SPLINE
SPL {X  -124.075, Y  +778.932, Z    +0.000, E1   -61.393, E3 +52956.323}
SPL {X  -150.653, Y  +735.257, Z    +0.000, E1   -50.160, E3 +52964.002}
SPL {X  -159.377, Y  +706.804, Z    +0.000, E1   -34.828, E3 +52965.646}
SPL {X  -162.134, Y  +688.425, Z    +0.000, E1   -19.100, E3 +52965.583}
SPL {X  -162.803, Y  +675.871, Z    +0.000, E1    -5.469, E3 +52965.766}
SPL {X  -162.820, Y  +671.500, Z    +0.000, E1    +0.000, E3 +52965.335}
SPL {X  -162.820, Y  +669.743, Z    +0.000, E1    +4.352, E3 +52965.130}
SPL {X  -162.820, Y  +665.917, Z    +0.000, E1   +15.272, E3 +52965.125}
SPL {X  -162.820, Y  +659.880, Z    +0.000, E1   +32.256, E3 +52965.036}
SPL {X  -162.820, Y  +652.069, Z    +0.000, E1   +49.663, E3 +52965.062}
SPL {X  -162.820, Y  +641.345, Z    +0.000, E1   +63.138, E3 +52965.160}
SPL {X  -162.820, Y  +620.039, Z    +0.000, E1   +75.979, E3 +52963.770}
SPL {X  -162.820, Y  +571.094, Z    +0.000, E1   +77.089, E3 +52978.948}
SPL {X  -157.487, Y  +339.169, Z    +0.000, E1   +76.425, E3 +53072.052}
SPL {X  -156.386, Y  +335.181, Z    +0.000, E1   +75.555, E3 +53084.113}
SPL {X  -152.710, Y  +324.020, Z    +0.000, E1   +75.365, E3 +53091.924}
SPL {X  -139.497, Y  +296.529, Z    +0.000, E1   +77.231, E3 +53085.495}
ENDSPLINE

SPLINE
SPL {X  -139.520, Y  +296.568, Z    +0.000, E1   +75.884, E3 +53098.143}
ENDSPLINE

SPLINE
SPL {X  -138.554, Y  +294.984, Z    +0.000, E1   +74.772, E3 +53108.024}
SPL {X  -137.186, Y  +292.805, Z    +0.000, E1   +73.993, E3 +53115.264}
SPL {X  -133.270, Y  +286.961, Z    +0.000, E1   +73.739, E3 +53119.977}
SPL {X  -129.057, Y  +281.230, Z    +0.000, E1   +73.118, E3 +53126.885}
SPL {X  -123.859, Y  +274.815, Z    +0.000, E1   +72.511, E3 +53133.269}
SPL {X  -121.018, Y  +271.573, Z    +0.000, E1   +72.049, E3 +53136.787}
SPL {X  -113.980, Y  +264.229, Z    +0.000, E1   +74.120, E3 +53132.365}
SPL {X   -56.216, Y  +227.692, Z    +0.000, E1   +56.267, E3 +53309.089}
ENDSPLINE

SPLINE
SPL {X  -126.995, Y  +278.604, Z    +0.000, E1   +59.937, E3 +53481.329}
SPL {X  -150.196, Y  +317.640, Z    +0.000, E1   +49.956, E3 +53489.784}
SPL {X  -157.261, Y  +338.316, Z    +0.000, E1   +40.017, E3 +53491.479}
SPL {X  -160.924, Y  +355.726, Z    +0.000, E1   +27.715, E3 +53491.920}
SPL {X  -162.423, Y  +369.141, Z    +0.000, E1   +15.207, E3 +53492.356}
SPL {X  -162.811, Y  +378.755, Z    +0.000, E1    +4.616, E3 +53492.270}
SPL {X  -162.820, Y  +382.684, Z    +0.000, E1    -0.227, E3 +53491.825}
SPL {X  -162.820, Y  +385.721, Z    +0.000, E1    -8.371, E3 +53491.640}
SPL {X  -162.820, Y  +388.532, Z    +0.000, E1   -16.412, E3 +53491.527}
SPL {X  -162.820, Y  +392.558, Z    +0.000, E1   -27.778, E3 +53491.616}
SPL {X  -162.820, Y  +400.474, Z    +0.000, E1   -46.251, E3 +53491.479}
SPL {X  -162.820, Y  +414.510, Z    +0.000, E1   -65.115, E3 +53490.922}
SPL {X  -162.820, Y  +465.064, Z    +0.000, E1   -76.269, E3 +53500.770}
SPL {X  -157.184, Y  +715.968, Z    +0.000, E1   -76.600, E3 +53596.728}
SPL {X  -156.461, Y  +718.560, Z    +0.000, E1   -75.553, E3 +53610.148}
SPL {X  -153.015, Y  +729.150, Z    +0.000, E1   -75.312, E3 +53618.237}
SPL {X  -149.053, Y  +739.025, Z    +0.000, E1   -74.952, E3 +53627.033}
SPL {X  -144.053, Y  +749.389, Z    +0.000, E1   -74.457, E3 +53637.024}
SPL {X  -139.539, Y  +757.399, Z    +0.000, E1   -73.892, E3 +53645.731}
SPL {X  -136.017, Y  +762.997, Z    +0.000, E1   -73.579, E3 +53650.913}
SPL {X  -133.089, Y  +767.296, Z    +0.000, E1   -73.251, E3 +53655.371}
SPL {X  -129.985, Y  +771.553, Z    +0.000, E1   -72.801, E3 +53660.365}
SPL {X  -126.581, Y  +775.909, Z    +0.000, E1   -72.426, E3 +53664.676}
SPL {X  -123.329, Y  +779.803, Z    +0.000, E1   -71.936, E3 +53669.058}
SPL {X  -119.291, Y  +784.315, Z    +0.000, E1   -72.148, E3 +53670.470}
SPL {X   -57.587, Y  +825.796, Z    +0.000, E1   -56.753, E3 +53824.233}
ENDSPLINE

SPLINE
SPL {X  -124.075, Y  +778.932, Z    +0.000, E1   -61.393, E3 +54017.862}
SPL {X  -150.653, Y  +735.257, Z    +0.000, E1   -50.160, E3 +54025.541}
SPL {X  -159.377, Y  +706.804, Z    +0.000, E1   -34.828, E3 +54027.184}
SPL {X  -162.134, Y  +688.425, Z    +0.000, E1   -19.100, E3 +54027.121}
SPL {X  -162.803, Y  +675.871, Z    +0.000, E1    -5.469, E3 +54027.305}
SPL {X  -162.820, Y  +671.500, Z    +0.000, E1    +0.000, E3 +54026.873}
SPL {X  -162.820, Y  +669.743, Z    +0.000, E1    +4.352, E3 +54026.669}
SPL {X  -162.820, Y  +665.917, Z    +0.000, E1   +15.272, E3 +54026.663}
SPL {X  -162.820, Y  +659.880, Z    +0.000, E1   +32.256, E3 +54026.575}
SPL {X  -162.820, Y  +652.069, Z    +0.000, E1   +49.663, E3 +54026.600}
SPL {X  -162.820, Y  +641.345, Z    +0.000, E1   +63.138, E3 +54026.698}
SPL {X  -162.820, Y  +620.039, Z    +0.000, E1   +75.979, E3 +54025.308}
SPL {X  -162.820, Y  +578.479, Z    +0.000, E1   +77.260, E3 +54037.579}
SPL {X  -162.820, Y  +557.052, Z    +0.000, E1   +76.772, E3 +54046.060}
SPL {X  -157.487, Y  +339.169, Z    +0.000, E1   +76.425, E3 +54133.591}
SPL {X  -156.386, Y  +335.181, Z    +0.000, E1   +75.555, E3 +54145.652}
SPL {X  -152.710, Y  +324.020, Z    +0.000, E1   +75.365, E3 +54153.462}
SPL {X  -139.497, Y  +296.529, Z    +0.000, E1   +77.231, E3 +54147.034}
ENDSPLINE

SPLINE
SPL {X  -139.792, Y  +297.022, Z    +0.000, E1   +76.273, E3 +54155.729}
ENDSPLINE

SPLINE
SPL {X  -138.933, Y  +295.600, Z    +0.000, E1   +75.173, E3 +54166.212}
SPL {X  -137.186, Y  +292.805, Z    +0.000, E1   +73.993, E3 +54176.802}
SPL {X  -133.270, Y  +286.961, Z    +0.000, E1   +73.739, E3 +54181.515}
SPL {X  -130.283, Y  +282.844, Z    +0.000, E1   +73.297, E3 +54186.407}
SPL {X  -126.880, Y  +278.461, Z    +0.000, E1   +72.855, E3 +54191.158}
SPL {X  -124.135, Y  +275.140, Z    +0.000, E1   +72.554, E3 +54194.286}
SPL {X  -121.687, Y  +272.322, Z    +0.000, E1   +72.100, E3 +54197.765}
SPL {X  -113.980, Y  +264.229, Z    +0.000, E1   +74.120, E3 +54193.903}
SPL {X   -56.216, Y  +227.692, Z    +0.000, E1   +56.267, E3 +54370.627}
ENDSPLINE

SPLINE
SPL {X  -126.995, Y  +278.604, Z    +0.000, E1   +59.937, E3 +54542.868}
SPL {X  -150.196, Y  +317.640, Z    +0.000, E1   +49.956, E3 +54551.323}
SPL {X  -157.261, Y  +338.316, Z    +0.000, E1   +40.017, E3 +54553.018}
SPL {X  -160.924, Y  +355.726, Z    +0.000, E1   +27.715, E3 +54553.459}
SPL {X  -162.423, Y  +369.141, Z    +0.000, E1   +15.207, E3 +54553.894}
SPL {X  -162.811, Y  +378.755, Z    +0.000, E1    +4.616, E3 +54553.808}
SPL {X  -162.820, Y  +382.684, Z    +0.000, E1    -0.227, E3 +54553.363}
SPL {X  -162.820, Y  +385.721, Z    +0.000, E1    -8.371, E3 +54553.179}
SPL {X  -162.820, Y  +388.532, Z    +0.000, E1   -16.412, E3 +54553.065}
SPL {X  -162.820, Y  +392.558, Z    +0.000, E1   -27.778, E3 +54553.154}
SPL {X  -162.820, Y  +400.474, Z    +0.000, E1   -46.251, E3 +54553.018}
SPL {X  -162.820, Y  +414.510, Z    +0.000, E1   -65.115, E3 +54552.461}
SPL {X  -162.820, Y  +465.064, Z    +0.000, E1   -76.269, E3 +54562.309}
SPL {X  -157.184, Y  +715.968, Z    +0.000, E1   -76.600, E3 +54658.266}
SPL {X  -156.461, Y  +718.560, Z    +0.000, E1   -75.553, E3 +54671.686}
SPL {X  -151.911, Y  +732.096, Z    +0.000, E1   -75.235, E3 +54682.240}
SPL {X  -146.569, Y  +744.407, Z    +0.000, E1   -74.677, E3 +54694.044}
SPL {X  -142.375, Y  +752.491, Z    +0.000, E1   -74.335, E3 +54701.072}
SPL {X  -139.539, Y  +757.399, Z    +0.000, E1   -73.892, E3 +54707.269}
SPL {X  -136.017, Y  +762.997, Z    +0.000, E1   -73.579, E3 +54712.452}
SPL {X  -133.089, Y  +767.296, Z    +0.000, E1   -73.251, E3 +54716.910}
SPL {X  -129.985, Y  +771.553, Z    +0.000, E1   -72.801, E3 +54721.904}
SPL {X  -126.581, Y  +775.909, Z    +0.000, E1   -72.426, E3 +54726.215}
SPL {X  -123.329, Y  +779.803, Z    +0.000, E1   -71.936, E3 +54730.597}
SPL {X  -119.291, Y  +784.315, Z    +0.000, E1   -72.148, E3 +54732.009}
SPL {X   -57.587, Y  +825.796, Z    +0.000, E1   -56.753, E3 +54885.771}
ENDSPLINE

SPLINE
SPL {X  -124.075, Y  +778.932, Z    +0.000, E1   -61.393, E3 +55079.400}
SPL {X  -147.028, Y  +743.450, Z    +0.000, E1   -53.078, E3 +55086.137}
SPL {X  -152.552, Y  +730.406, Z    +0.000, E1   -48.136, E3 +55087.555}
SPL {X  -159.377, Y  +706.804, Z    +0.000, E1   -34.828, E3 +55088.723}
SPL {X  -162.134, Y  +688.425, Z    +0.000, E1   -19.100, E3 +55088.659}
SPL {X  -162.803, Y  +675.871, Z    +0.000, E1    -5.469, E3 +55088.843}
SPL {X  -162.820, Y  +671.500, Z    +0.000, E1    +0.000, E3 +55088.411}
SPL {X  -162.820, Y  +669.743, Z    +0.000, E1    +4.352, E3 +55088.207}
SPL {X  -162.820, Y  +665.917, Z    +0.000, E1   +15.272, E3 +55088.202}
SPL {X  -162.820, Y  +661.245, Z    +0.000, E1   +28.879, E3 +55088.043}
SPL {X  -162.820, Y  +654.015, Z    +0.000, E1   +45.814, E3 +55088.190}
SPL {X  -162.820, Y  +641.345, Z    +0.000, E1   +63.138, E3 +55088.237}
SPL {X  -162.820, Y  +620.039, Z    +0.000, E1   +75.979, E3 +55086.847}
SPL {X  -162.820, Y  +571.094, Z    +0.000, E1   +77.089, E3 +55102.025}
SPL {X  -157.487, Y  +339.169, Z    +0.000, E1   +76.425, E3 +55195.129}
SPL {X  -156.386, Y  +335.181, Z    +0.000, E1   +75.555, E3 +55207.190}
SPL {X  -152.710, Y  +324.020, Z    +0.000, E1   +75.365, E3 +55215.000}
SPL {X  -139.497, Y  +296.529, Z    +0.000, E1   +77.231, E3 +55208.572}
ENDSPLINE

SPLINE
SPL {X  -139.792, Y  +297.022, Z    +0.000, E1   +76.273, E3 +55217.267}
ENDSPLINE

SPLINE
SPL {X  -138.933, Y  +295.600, Z    +0.000, E1   +75.173, E3 +55227.750}
SPL {X  -137.186, Y  +292.805, Z    +0.000, E1   +73.993, E3 +55238.340}
SPL {X  -133.270, Y  +286.961, Z    +0.000, E1   +73.739, E3 +55243.054}
SPL {X  -130.283, Y  +282.844, Z    +0.000, E1   +73.297, E3 +55247.946}
SPL {X  -126.880, Y  +278.461, Z    +0.000, E1   +72.855, E3 +55252.696}
SPL {X  -123.363, Y  +274.237, Z    +0.000, E1   +72.376, E3 +55257.178}
SPL {X  -121.018, Y  +271.573, Z    +0.000, E1   +72.049, E3 +55259.863}
SPL {X  -113.980, Y  +264.229, Z    +0.000, E1   +74.120, E3 +55255.442}
SPL {X   -56.216, Y  +227.692, Z    +0.000, E1   +56.267, E3 +55432.166}
ENDSPLINE

SPLINE
SPL {X  -126.995, Y  +278.604, Z    +0.000, E1   +59.937, E3 +55604.406}
SPL {X  -150.196, Y  +317.640, Z    +0.000, E1   +49.956, E3 +55612.861}
SPL {X  -157.261, Y  +338.316, Z    +0.000, E1   +40.017, E3 +55614.556}
SPL {X  -160.924, Y  +355.726, Z    +0.000, E1   +27.715, E3 +55614.997}
SPL {X  -162.423, Y  +369.141, Z    +0.000, E1   +15.207, E3 +55615.432}
SPL {X  -162.811, Y  +378.755, Z    +0.000, E1    +4.616, E3 +55615.347}
SPL {X  -162.820, Y  +382.684, Z    +0.000, E1    -0.227, E3 +55614.902}
SPL {X  -162.820, Y  +385.721, Z    +0.000, E1    -8.371, E3 +55614.717}
SPL {X  -162.820, Y  +388.532, Z    +0.000, E1   -16.412, E3 +55614.604}
SPL {X  -162.820, Y  +392.558, Z    +0.000, E1   -27.778, E3 +55614.692}
SPL {X  -162.820, Y  +400.474, Z    +0.000, E1   -46.251, E3 +55614.556}
SPL {X  -162.820, Y  +414.510, Z    +0.000, E1   -65.115, E3 +55613.999}
SPL {X  -162.820, Y  +465.064, Z    +0.000, E1   -76.269, E3 +55623.847}
SPL {X  -157.184, Y  +715.968, Z    +0.000, E1   -76.600, E3 +55719.805}
SPL {X  -156.461, Y  +718.560, Z    +0.000, E1   -75.553, E3 +55733.225}
SPL {X  -151.911, Y  +732.096, Z    +0.000, E1   -75.235, E3 +55743.779}
SPL {X  -146.569, Y  +744.407, Z    +0.000, E1   -74.677, E3 +55755.583}
SPL {X  -142.375, Y  +752.491, Z    +0.000, E1   -74.335, E3 +55762.610}
SPL {X  -139.539, Y  +757.399, Z    +0.000, E1   -73.892, E3 +55768.808}
SPL {X  -136.017, Y  +762.997, Z    +0.000, E1   -73.579, E3 +55773.990}
SPL {X  -133.089, Y  +767.296, Z    +0.000, E1   -73.251, E3 +55778.448}
SPL {X  -129.985, Y  +771.553, Z    +0.000, E1   -72.801, E3 +55783.442}
SPL {X  -126.581, Y  +775.909, Z    +0.000, E1   -72.426, E3 +55787.753}
SPL {X  -123.329, Y  +779.803, Z    +0.000, E1   -71.936, E3 +55792.135}
SPL {X  -119.291, Y  +784.315, Z    +0.000, E1   -72.148, E3 +55793.547}
SPL {X   -57.587, Y  +825.796, Z    +0.000, E1   -56.753, E3 +55947.309}
ENDSPLINE

SPLINE
SPL {X  -124.075, Y  +778.932, Z    +0.000, E1   -61.393, E3 +56140.938}
SPL {X  -147.028, Y  +743.450, Z    +0.000, E1   -53.078, E3 +56147.676}
SPL {X  -152.552, Y  +730.406, Z    +0.000, E1   -48.136, E3 +56149.093}
SPL {X  -159.377, Y  +706.804, Z    +0.000, E1   -34.828, E3 +56150.261}
SPL {X  -162.134, Y  +688.425, Z    +0.000, E1   -19.100, E3 +56150.198}
SPL {X  -162.803, Y  +675.871, Z    +0.000, E1    -5.469, E3 +56150.382}
SPL {X  -162.820, Y  +671.500, Z    +0.000, E1    +0.000, E3 +56149.950}
SPL {X  -162.820, Y  +669.743, Z    +0.000, E1    +4.352, E3 +56149.746}
SPL {X  -162.820, Y  +665.917, Z    +0.000, E1   +15.272, E3 +56149.740}
SPL {X  -162.820, Y  +661.245, Z    +0.000, E1   +28.879, E3 +56149.581}
SPL {X  -162.820, Y  +654.015, Z    +0.000, E1   +45.814, E3 +56149.728}
SPL {X  -162.820, Y  +641.345, Z    +0.000, E1   +63.138, E3 +56149.775}
SPL {X  -162.820, Y  +620.039, Z    +0.000, E1   +75.979, E3 +56148.385}
SPL {X  -162.820, Y  +571.094, Z    +0.000, E1   +77.089, E3 +56163.564}
SPL {X  -157.487, Y  +339.169, Z    +0.000, E1   +76.425, E3 +56256.668}
SPL {X  -156.386, Y  +335.181, Z    +0.000, E1   +75.555, E3 +56268.729}
SPL {X  -152.710, Y  +324.020, Z    +0.000, E1   +75.365, E3 +56276.539}
SPL {X  -139.497, Y  +296.529, Z    +0.000, E1   +77.231, E3 +56270.111}
ENDSPLINE

SPLINE
SPL {X  -139.792, Y  +297.022, Z    +0.000, E1   +76.273, E3 +56278.806}
ENDSPLINE

SPLINE
SPL {X  -138.933, Y  +295.600, Z    +0.000, E1   +75.173, E3 +56289.289}
SPL {X  -137.186, Y  +292.805, Z    +0.000, E1   +73.993, E3 +56299.879}
SPL {X  -133.270, Y  +286.961, Z    +0.000, E1   +73.739, E3 +56304.592}
SPL {X  -130.283, Y  +282.844, Z    +0.000, E1   +73.297, E3 +56309.484}
SPL {X  -127.795, Y  +279.610, Z    +0.000, E1   +72.860, E3 +56313.614}
SPL {X  -124.650, Y  +275.749, Z    +0.000, E1   +72.674, E3 +56316.533}
SPL {X  -121.687, Y  +272.322, Z    +0.000, E1   +72.100, E3 +56320.842}
SPL {X  -113.980, Y  +264.229, Z    +0.000, E1   +74.120, E3 +56316.980}
SPL {X   -56.216, Y  +227.692, Z    +0.000, E1   +56.267, E3 +56493.704}
ENDSPLINE

SPLINE
SPL {X  -126.995, Y  +278.604, Z    +0.000, E1   +59.937, E3 +56665.945}
SPL {X  -150.196, Y  +317.640, Z    +0.000, E1   +49.956, E3 +56674.400}
SPL {X  -157.261, Y  +338.316, Z    +0.000, E1   +40.017, E3 +56676.095}
SPL {X  -160.924, Y  +355.726, Z    +0.000, E1   +27.715, E3 +56676.535}
SPL {X  -162.423, Y  +369.141, Z    +0.000, E1   +15.207, E3 +56676.971}
SPL {X  -162.811, Y  +378.755, Z    +0.000, E1    +4.616, E3 +56676.885}
SPL {X  -162.820, Y  +382.684, Z    +0.000, E1    -0.227, E3 +56676.440}
SPL {X  -162.820, Y  +387.227, Z    +0.000, E1   -12.320, E3 +56676.195}
SPL {X  -162.820, Y  +392.558, Z    +0.000, E1   -27.778, E3 +56676.231}
SPL {X  -162.820, Y  +400.474, Z    +0.000, E1   -46.251, E3 +56676.095}
SPL {X  -162.820, Y  +414.510, Z    +0.000, E1   -65.115, E3 +56675.538}
SPL {X  -162.820, Y  +465.064, Z    +0.000, E1   -76.269, E3 +56685.386}
SPL {X  -157.184, Y  +715.968, Z    +0.000, E1   -76.600, E3 +56781.343}
SPL {X  -156.461, Y  +718.560, Z    +0.000, E1   -75.553, E3 +56794.763}
SPL {X  -153.015, Y  +729.150, Z    +0.000, E1   -75.312, E3 +56802.852}
SPL {X  -149.053, Y  +739.025, Z    +0.000, E1   -74.952, E3 +56811.648}
SPL {X  -145.525, Y  +746.527, Z    +0.000, E1   -74.526, E3 +56819.441}
SPL {X  -142.375, Y  +752.491, Z    +0.000, E1   -74.335, E3 +56824.149}
SPL {X  -139.539, Y  +757.399, Z    +0.000, E1   -73.892, E3 +56830.346}
SPL {X  -136.017, Y  +762.997, Z    +0.000, E1   -73.579, E3 +56835.529}
SPL {X  -133.089, Y  +767.296, Z    +0.000, E1   -73.251, E3 +56839.987}
SPL {X  -129.985, Y  +771.553, Z    +0.000, E1   -72.801, E3 +56844.981}
SPL {X  -126.581, Y  +775.909, Z    +0.000, E1   -72.426, E3 +56849.292}
SPL {X  -123.329, Y  +779.803, Z    +0.000, E1   -71.936, E3 +56853.674}
SPL {X  -119.291, Y  +784.315, Z    +0.000, E1   -72.148, E3 +56855.085}
SPL {X   -57.587, Y  +825.796, Z    +0.000, E1   -56.753, E3 +57008.848}
ENDSPLINE

SPLINE
SPL {X  -124.075, Y  +778.932, Z    +0.000, E1   -61.393, E3 +57202.477}
SPL {X  -150.653, Y  +735.257, Z    +0.000, E1   -50.160, E3 +57210.156}
SPL {X  -159.377, Y  +706.804, Z    +0.000, E1   -34.828, E3 +57211.800}
SPL {X  -162.134, Y  +688.425, Z    +0.000, E1   -19.100, E3 +57211.736}
SPL {X  -162.803, Y  +675.871, Z    +0.000, E1    -5.469, E3 +57211.920}
SPL {X  -162.820, Y  +671.500, Z    +0.000, E1    +0.000, E3 +57211.488}
SPL {X  -162.820, Y  +669.743, Z    +0.000, E1    +4.352, E3 +57211.284}
SPL {X  -162.820, Y  +665.917, Z    +0.000, E1   +15.272, E3 +57211.279}
SPL {X  -162.820, Y  +661.245, Z    +0.000, E1   +28.879, E3 +57211.120}
SPL {X  -162.820, Y  +654.015, Z    +0.000, E1   +45.814, E3 +57211.267}
SPL {X  -162.820, Y  +641.345, Z    +0.000, E1   +63.138, E3 +57211.314}
SPL {X  -162.820, Y  +620.039, Z    +0.000, E1   +75.979, E3 +57209.924}
SPL {X  -162.820, Y  +571.094, Z    +0.000, E1   +77.089, E3 +57225.102}
SPL {X  -157.487, Y  +339.169, Z    +0.000, E1   +76.425, E3 +57318.206}
SPL {X  -156.386, Y  +335.181, Z    +0.000, E1   +75.555, E3 +57330.267}
SPL {X  -152.710, Y  +324.020, Z    +0.000, E1   +75.365, E3 +57338.077}
SPL {X  -139.497, Y  +296.529, Z    +0.000, E1   +77.231, E3 +57331.649}
ENDSPLINE

SPLINE
SPL {X  -139.792, Y  +297.022, Z    +0.000, E1   +76.273, E3 +57340.344}
ENDSPLINE

SPLINE
SPL {X  -138.933, Y  +295.600, Z    +0.000, E1   +75.173, E3 +57350.827}
SPL {X  -137.186, Y  +292.805, Z    +0.000, E1   +73.993, E3 +57361.417}
SPL {X  -133.270, Y  +286.961, Z    +0.000, E1   +73.739, E3 +57366.131}
SPL {X  -130.283, Y  +282.844, Z    +0.000, E1   +73.297, E3 +57371.023}
SPL {X  -127.795, Y  +279.610, Z    +0.000, E1   +72.860, E3 +57375.153}
SPL {X  -124.650, Y  +275.749, Z    +0.000, E1   +72.674, E3 +57378.071}
SPL {X  -121.687, Y  +272.322, Z    +0.000, E1   +72.100, E3 +57382.381}
SPL {X  -113.980, Y  +264.229, Z    +0.000, E1   +74.120, E3 +57378.519}
SPL {X   -56.216, Y  +227.692, Z    +0.000, E1   +56.267, E3 +57555.243}
ENDSPLINE

SPLINE
SPL {X  -126.995, Y  +278.604, Z    +0.000, E1   +59.937, E3 +57727.483}
SPL {X  -150.196, Y  +317.640, Z    +0.000, E1   +49.956, E3 +57735.938}
SPL {X  -157.261, Y  +338.316, Z    +0.000, E1   +40.017, E3 +57737.633}
SPL {X  -160.924, Y  +355.726, Z    +0.000, E1   +27.715, E3 +57738.074}
SPL {X  -162.423, Y  +369.141, Z    +0.000, E1   +15.207, E3 +57738.509}
SPL {X  -162.811, Y  +378.755, Z    +0.000, E1    +4.616, E3 +57738.424}
SPL {X  -162.820, Y  +382.684, Z    +0.000, E1    -0.227, E3 +57737.978}
SPL {X  -162.820, Y  +387.227, Z    +0.000, E1   -12.320, E3 +57737.733}
SPL {X  -162.820, Y  +392.558, Z    +0.000, E1   -27.778, E3 +57737.769}
SPL {X  -162.820, Y  +400.474, Z    +0.000, E1   -46.251, E3 +57737.633}
SPL {X  -162.820, Y  +414.510, Z    +0.000, E1   -65.115, E3 +57737.076}
SPL {X  -162.820, Y  +465.064, Z    +0.000, E1   -76.269, E3 +57746.924}
SPL {X  -158.097, Y  +712.432, Z    +0.000, E1   -77.677, E3 +57829.312}
SPL {X  -156.557, Y  +718.224, Z    +0.000, E1   -75.715, E3 +57854.448}
SPL {X  -151.911, Y  +732.096, Z    +0.000, E1   -75.235, E3 +57866.856}
SPL {X  -146.569, Y  +744.407, Z    +0.000, E1   -74.677, E3 +57878.660}
SPL {X  -142.375, Y  +752.491, Z    +0.000, E1   -74.335, E3 +57885.687}
SPL {X  -139.539, Y  +757.399, Z    +0.000, E1   -73.892, E3 +57891.885}
SPL {X  -136.017, Y  +762.997, Z    +0.000, E1   -73.579, E3 +57897.067}
SPL {X  -133.089, Y  +767.296, Z    +0.000, E1   -73.251, E3 +57901.525}
SPL {X  -129.985, Y  +771.553, Z    +0.000, E1   -72.801, E3 +57906.519}
SPL {X  -126.581, Y  +775.909, Z    +0.000, E1   -72.426, E3 +57910.830}
SPL {X  -123.329, Y  +779.803, Z    +0.000, E1   -71.936, E3 +57915.212}
SPL {X  -119.291, Y  +784.315, Z    +0.000, E1   -72.148, E3 +57916.624}
SPL {X   -57.587, Y  +825.796, Z    +0.000, E1   -56.753, E3 +58070.386}
ENDSPLINE

SPLINE
SPL {X  -124.075, Y  +778.932, Z    +0.000, E1   -61.393, E3 +58264.015}
SPL {X  -150.653, Y  +735.257, Z    +0.000, E1   -50.160, E3 +58271.695}
SPL {X  -159.377, Y  +706.804, Z    +0.000, E1   -34.828, E3 +58273.338}
SPL {X  -162.134, Y  +688.425, Z    +0.000, E1   -19.100, E3 +58273.275}
SPL {X  -162.803, Y  +675.871, Z    +0.000, E1    -5.469, E3 +58273.459}
SPL {X  -162.820, Y  +671.500, Z    +0.000, E1    +0.000, E3 +58273.027}
SPL {X  -162.820, Y  +669.743, Z    +0.000, E1    +4.352, E3 +58272.822}
SPL {X  -162.820, Y  +665.917, Z    +0.000, E1   +15.272, E3 +58272.817}
SPL {X  -162.820, Y  +661.245, Z    +0.000, E1   +28.879, E3 +58272.658}
SPL {X  -162.820, Y  +654.015, Z    +0.000, E1   +45.814, E3 +58272.805}
SPL {X  -162.820, Y  +641.345, Z    +0.000, E1   +63.138, E3 +58272.852}
SPL {X  -162.820, Y  +620.039, Z    +0.000, E1   +75.979, E3 +58271.462}
SPL {X  -162.820, Y  +571.094, Z    +0.000, E1   +77.089, E3 +58286.641}
SPL {X  -157.487, Y  +339.169, Z    +0.000, E1   +76.425, E3 +58379.745}
SPL {X  -156.386, Y  +335.181, Z    +0.000, E1   +75.555, E3 +58391.805}
SPL {X  -152.710, Y  +324.020, Z    +0.000, E1   +75.365, E3 +58399.616}
SPL {X  -139.497, Y  +296.529, Z    +0.000, E1   +77.231, E3 +58393.188}
ENDSPLINE

SPLINE
SPL {X  -139.792, Y  +297.022, Z    +0.000, E1   +76.273, E3 +58401.883}
ENDSPLINE

SPLINE
SPL {X  -138.933, Y  +295.600, Z    +0.000, E1   +75.173, E3 +58412.365}
SPL {X  -137.186, Y  +292.805, Z    +0.000, E1   +73.993, E3 +58422.956}
SPL {X  -133.270, Y  +286.961, Z    +0.000, E1   +73.739, E3 +58427.669}
SPL {X  -130.283, Y  +282.844, Z    +0.000, E1   +73.297, E3 +58432.561}
SPL {X  -127.795, Y  +279.610, Z    +0.000, E1   +72.860, E3 +58436.691}
SPL {X  -124.650, Y  +275.749, Z    +0.000, E1   +72.674, E3 +58439.610}
SPL {X  -121.687, Y  +272.322, Z    +0.000, E1   +72.100, E3 +58443.919}
SPL {X  -113.980, Y  +264.229, Z    +0.000, E1   +74.120, E3 +58440.057}
SPL {X   -56.216, Y  +227.692, Z    +0.000, E1   +56.267, E3 +58616.781}
ENDSPLINE

SPLINE
SPL {X  -126.995, Y  +278.604, Z    +0.000, E1   +59.937, E3 +58789.021}
SPL {X  -150.196, Y  +317.640, Z    +0.000, E1   +49.956, E3 +58797.477}
SPL {X  -157.261, Y  +338.316, Z    +0.000, E1   +40.017, E3 +58799.172}
SPL {X  -160.924, Y  +355.726, Z    +0.000, E1   +27.715, E3 +58799.612}
SPL {X  -162.423, Y  +369.141, Z    +0.000, E1   +15.207, E3 +58800.048}
SPL {X  -162.811, Y  +378.755, Z    +0.000, E1    +4.616, E3 +58799.962}
SPL {X  -162.820, Y  +382.684, Z    +0.000, E1    -0.227, E3 +58799.517}
SPL {X  -162.820, Y  +387.227, Z    +0.000, E1   -12.320, E3 +58799.272}
SPL {X  -162.820, Y  +392.558, Z    +0.000, E1   -27.778, E3 +58799.308}
SPL {X  -162.820, Y  +400.474, Z    +0.000, E1   -46.251, E3 +58799.172}
SPL {X  -162.820, Y  +414.510, Z    +0.000, E1   -65.115, E3 +58798.615}
SPL {X  -162.820, Y  +465.064, Z    +0.000, E1   -76.269, E3 +58808.463}
SPL {X  -158.097, Y  +712.432, Z    +0.000, E1   -77.677, E3 +58890.850}
SPL {X  -156.557, Y  +718.224, Z    +0.000, E1   -75.715, E3 +58915.987}
SPL {X  -151.911, Y  +732.096, Z    +0.000, E1   -75.235, E3 +58928.394}
SPL {X  -146.569, Y  +744.407, Z    +0.000, E1   -74.677, E3 +58940.198}
SPL {X  -142.375, Y  +752.491, Z    +0.000, E1   -74.335, E3 +58947.226}
SPL {X  -139.539, Y  +757.399, Z    +0.000, E1   -73.892, E3 +58953.423}
SPL {X  -136.017, Y  +762.997, Z    +0.000, E1   -73.579, E3 +58958.606}
SPL {X  -133.089, Y  +767.296, Z    +0.000, E1   -73.251, E3 +58963.064}
SPL {X  -129.985, Y  +771.553, Z    +0.000, E1   -72.801, E3 +58968.057}
SPL {X  -126.581, Y  +775.909, Z    +0.000, E1   -72.426, E3 +58972.369}
SPL {X  -123.329, Y  +779.803, Z    +0.000, E1   -71.936, E3 +58976.750}
SPL {X  -119.291, Y  +784.315, Z    +0.000, E1   -72.148, E3 +58978.162}
SPL {X   -57.587, Y  +825.796, Z    +0.000, E1   -56.753, E3 +59131.925}
ENDSPLINE

SPLINE
SPL {X  -124.075, Y  +778.932, Z    +0.000, E1   -61.393, E3 +59325.554}
SPL {X  -150.653, Y  +735.257, Z    +0.000, E1   -50.160, E3 +59333.233}
SPL {X  -159.377, Y  +706.804, Z    +0.000, E1   -34.828, E3 +59334.876}
SPL {X  -162.134, Y  +688.425, Z    +0.000, E1   -19.100, E3 +59334.813}
SPL {X  -162.803, Y  +675.871, Z    +0.000, E1    -5.469, E3 +59334.997}
SPL {X  -162.820, Y  +671.500, Z    +0.000, E1    +0.000, E3 +59334.565}
SPL {X  -162.820, Y  +669.743, Z    +0.000, E1    +4.352, E3 +59334.361}
SPL {X  -162.820, Y  +665.917, Z    +0.000, E1   +15.272, E3 +59334.355}
SPL {X  -162.820, Y  +661.245, Z    +0.000, E1   +28.879, E3 +59334.197}
SPL {X  -162.820, Y  +654.015, Z    +0.000, E1   +45.814, E3 +59334.344}
SPL {X  -162.820, Y  +641.345, Z    +0.000, E1   +63.138, E3 +59334.391}
SPL {X  -162.820, Y  +620.039, Z    +0.000, E1   +75.979, E3 +59333.001}
SPL {X  -162.820, Y  +578.479, Z    +0.000, E1   +77.260, E3 +59345.271}
SPL {X  -162.820, Y  +557.052, Z    +0.000, E1   +76.772, E3 +59353.753}
SPL {X  -157.487, Y  +339.169, Z    +0.000, E1   +76.425, E3 +59441.283}
SPL {X  -156.386, Y  +335.181, Z    +0.000, E1   +75.555, E3 +59453.344}
SPL {X  -152.710, Y  +324.020, Z    +0.000, E1   +75.365, E3 +59461.154}
SPL {X  -139.497, Y  +296.529, Z    +0.000, E1   +77.231, E3 +59454.726}
ENDSPLINE

SPLINE
SPL {X  -139.792, Y  +297.022, Z    +0.000, E1   +76.273, E3 +59463.421}
ENDSPLINE

SPLINE
SPL {X  -138.933, Y  +295.600, Z    +0.000, E1   +75.173, E3 +59473.904}
SPL {X  -137.186, Y  +292.805, Z    +0.000, E1   +73.993, E3 +59484.494}
SPL {X  -133.270, Y  +286.961, Z    +0.000, E1   +73.739, E3 +59489.208}
SPL {X  -130.283, Y  +282.844, Z    +0.000, E1   +73.297, E3 +59494.100}
SPL {X  -126.880, Y  +278.461, Z    +0.000, E1   +72.855, E3 +59498.850}
SPL {X  -124.135, Y  +275.140, Z    +0.000, E1   +72.554, E3 +59501.979}
SPL {X  -121.687, Y  +272.322, Z    +0.000, E1   +72.100, E3 +59505.457}
SPL {X  -113.980, Y  +264.229, Z    +0.000, E1   +74.120, E3 +59501.596}
SPL {X   -56.216, Y  +227.692, Z    +0.000, E1   +56.267, E3 +59678.320}
ENDSPLINE

SPLINE
SPL {X  -126.995, Y  +278.604, Z    +0.000, E1   +59.937, E3 +59850.560}
SPL {X  -150.196, Y  +317.640, Z    +0.000, E1   +49.956, E3 +59859.015}
SPL {X  -157.261, Y  +338.316, Z    +0.000, E1   +40.017, E3 +59860.710}
SPL {X  -160.924, Y  +355.726, Z    +0.000, E1   +27.715, E3 +59861.151}
SPL {X  -162.423, Y  +369.141, Z    +0.000, E1   +15.207, E3 +59861.586}
SPL {X  -162.811, Y  +378.755, Z    +0.000, E1    +4.616, E3 +59861.501}
SPL {X  -162.820, Y  +382.684, Z    +0.000, E1    -0.227, E3 +59861.055}
SPL {X  -162.820, Y  +385.721, Z    +0.000, E1    -8.371, E3 +59860.871}
SPL {X  -162.820, Y  +388.532, Z    +0.000, E1   -16.412, E3 +59860.757}
SPL {X  -162.820, Y  +392.558, Z    +0.000, E1   -27.778, E3 +59860.846}
SPL {X  -162.820, Y  +400.474, Z    +0.000, E1   -46.251, E3 +59860.710}
SPL {X  -162.820, Y  +414.510, Z    +0.000, E1   -65.115, E3 +59860.153}
SPL {X  -162.820, Y  +465.064, Z    +0.000, E1   -76.269, E3 +59870.001}
SPL {X  -157.184, Y  +715.968, Z    +0.000, E1   -76.600, E3 +59965.959}
SPL {X  -156.461, Y  +718.560, Z    +0.000, E1   -75.553, E3 +59979.378}
SPL {X  -153.015, Y  +729.150, Z    +0.000, E1   -75.312, E3 +59987.468}
SPL {X  -149.053, Y  +739.025, Z    +0.000, E1   -74.952, E3 +59996.263}
SPL {X  -144.053, Y  +749.389, Z    +0.000, E1   -74.457, E3 +60006.255}
SPL {X  -139.539, Y  +757.399, Z    +0.000, E1   -73.892, E3 +60014.962}
SPL {X  -136.017, Y  +762.997, Z    +0.000, E1   -73.579, E3 +60020.144}
SPL {X  -133.089, Y  +767.296, Z    +0.000, E1   -73.251, E3 +60024.602}
SPL {X  -129.985, Y  +771.553, Z    +0.000, E1   -72.801, E3 +60029.596}
SPL {X  -126.581, Y  +775.909, Z    +0.000, E1   -72.426, E3 +60033.907}
SPL {X  -123.329, Y  +779.803, Z    +0.000, E1   -71.936, E3 +60038.289}
SPL {X  -119.291, Y  +784.315, Z    +0.000, E1   -72.148, E3 +60039.701}
SPL {X   -57.587, Y  +825.796, Z    +0.000, E1   -56.753, E3 +60193.463}
ENDSPLINE

SPLINE
SPL {X  -124.075, Y  +778.932, Z    +0.000, E1   -61.393, E3 +60387.092}
SPL {X  -147.028, Y  +743.450, Z    +0.000, E1   -53.078, E3 +60393.829}
SPL {X  -152.552, Y  +730.406, Z    +0.000, E1   -48.136, E3 +60395.247}
SPL {X  -159.377, Y  +706.804, Z    +0.000, E1   -34.828, E3 +60396.415}
SPL {X  -162.134, Y  +688.425, Z    +0.000, E1   -19.100, E3 +60396.352}
SPL {X  -162.803, Y  +675.871, Z    +0.000, E1    -5.469, E3 +60396.536}
SPL {X  -162.820, Y  +671.500, Z    +0.000, E1    +0.000, E3 +60396.104}
SPL {X  -162.820, Y  +669.743, Z    +0.000, E1    +4.352, E3 +60395.899}
SPL {X  -162.820, Y  +665.917, Z    +0.000, E1   +15.272, E3 +60395.894}
SPL {X  -162.820, Y  +661.245, Z    +0.000, E1   +28.879, E3 +60395.735}
SPL {X  -162.820, Y  +654.015, Z    +0.000, E1   +45.814, E3 +60395.882}
SPL {X  -162.820, Y  +641.345, Z    +0.000, E1   +63.138, E3 +60395.929}
SPL {X  -162.820, Y  +620.039, Z    +0.000, E1   +75.979, E3 +60394.539}
SPL {X  -162.820, Y  +571.094, Z    +0.000, E1   +77.089, E3 +60409.718}
SPL {X  -157.487, Y  +339.169, Z    +0.000, E1   +76.425, E3 +60502.822}
SPL {X  -156.386, Y  +335.181, Z    +0.000, E1   +75.555, E3 +60514.882}
SPL {X  -152.710, Y  +324.020, Z    +0.000, E1   +75.365, E3 +60522.693}
SPL {X  -139.497, Y  +296.529, Z    +0.000, E1   +77.231, E3 +60516.264}
ENDSPLINE

SPLINE
SPL {X  -139.792, Y  +297.022, Z    +0.000, E1   +76.273, E3 +60524.960}
ENDSPLINE

SPLINE
SPL {X  -138.933, Y  +295.600, Z    +0.000, E1   +75.173, E3 +60535.442}
SPL {X  -137.186, Y  +292.805, Z    +0.000, E1   +73.993, E3 +60546.033}
SPL {X  -133.270, Y  +286.961, Z    +0.000, E1   +73.739, E3 +60550.746}
SPL {X  -130.283, Y  +282.844, Z    +0.000, E1   +73.297, E3 +60555.638}
SPL {X  -126.880, Y  +278.461, Z    +0.000, E1   +72.855, E3 +60560.389}
SPL {X  -123.363, Y  +274.237, Z    +0.000, E1   +72.376, E3 +60564.871}
SPL {X  -121.018, Y  +271.573, Z    +0.000, E1   +72.049, E3 +60567.556}
SPL {X  -113.980, Y  +264.229, Z    +0.000, E1   +74.120, E3 +60563.134}
SPL {X   -56.216, Y  +227.692, Z    +0.000, E1   +56.267, E3 +60739.858}
ENDSPLINE

SPLINE
SPL {X  -126.995, Y  +278.604, Z    +0.000, E1   +59.937, E3 +60912.098}
SPL {X  -150.196, Y  +317.640, Z    +0.000, E1   +49.956, E3 +60920.553}
SPL {X  -157.261, Y  +338.316, Z    +0.000, E1   +40.017, E3 +60922.249}
SPL {X  -160.924, Y  +355.726, Z    +0.000, E1   +27.715, E3 +60922.689}
SPL {X  -162.423, Y  +369.141, Z    +0.000, E1   +15.207, E3 +60923.125}
SPL {X  -162.811, Y  +378.755, Z    +0.000, E1    +4.616, E3 +60923.039}
SPL {X  -162.820, Y  +382.684, Z    +0.000, E1    -0.227, E3 +60922.594}
SPL {X  -162.820, Y  +387.227, Z    +0.000, E1   -12.320, E3 +60922.349}
SPL {X  -162.820, Y  +392.558, Z    +0.000, E1   -27.778, E3 +60922.385}
SPL {X  -162.820, Y  +398.468, Z    +0.000, E1   -42.446, E3 +60922.235}
SPL {X  -162.820, Y  +404.415, Z    +0.000, E1   -53.236, E3 +60922.274}
SPL {X  -162.820, Y  +414.510, Z    +0.000, E1   -65.115, E3 +60921.692}
SPL {X  -162.820, Y  +465.064, Z    +0.000, E1   -76.269, E3 +60931.540}
SPL {X  -157.184, Y  +715.968, Z    +0.000, E1   -76.600, E3 +61027.497}
SPL {X  -156.461, Y  +718.560, Z    +0.000, E1   -75.553, E3 +61040.917}
SPL {X  -151.911, Y  +732.096, Z    +0.000, E1   -75.235, E3 +61051.471}
SPL {X  -146.569, Y  +744.407, Z    +0.000, E1   -74.677, E3 +61063.275}
SPL {X  -142.375, Y  +752.491, Z    +0.000, E1   -74.335, E3 +61070.303}
SPL {X  -139.539, Y  +757.399, Z    +0.000, E1   -73.892, E3 +61076.500}
SPL {X  -136.017, Y  +762.997, Z    +0.000, E1   -73.579, E3 +61081.683}
SPL {X  -133.089, Y  +767.296, Z    +0.000, E1   -73.251, E3 +61086.141}
SPL {X  -129.985, Y  +771.553, Z    +0.000, E1   -72.801, E3 +61091.134}
SPL {X  -126.581, Y  +775.909, Z    +0.000, E1   -72.426, E3 +61095.446}
SPL {X  -123.329, Y  +779.803, Z    +0.000, E1   -71.936, E3 +61099.827}
SPL {X  -119.291, Y  +784.315, Z    +0.000, E1   -72.148, E3 +61101.239}
SPL {X   -57.587, Y  +825.796, Z    +0.000, E1   -56.753, E3 +61255.002}
ENDSPLINE

SPLINE
SPL {X  -124.075, Y  +778.932, Z    +0.000, E1   -61.393, E3 +61448.631}
SPL {X  -147.028, Y  +743.450, Z    +0.000, E1   -53.078, E3 +61455.368}
SPL {X  -152.552, Y  +730.406, Z    +0.000, E1   -48.136, E3 +61456.786}
SPL {X  -159.377, Y  +706.804, Z    +0.000, E1   -34.828, E3 +61457.953}
SPL {X  -162.134, Y  +688.425, Z    +0.000, E1   -19.100, E3 +61457.890}
SPL {X  -162.803, Y  +675.871, Z    +0.000, E1    -5.469, E3 +61458.074}
SPL {X  -162.820, Y  +671.500, Z    +0.000, E1    +0.000, E3 +61457.642}
SPL {X  -162.820, Y  +669.743, Z    +0.000, E1    +4.352, E3 +61457.438}
SPL {X  -162.820, Y  +665.917, Z    +0.000, E1   +15.272, E3 +61457.432}
SPL {X  -162.820, Y  +661.245, Z    +0.000, E1   +28.879, E3 +61457.274}
SPL {X  -162.820, Y  +654.015, Z    +0.000, E1   +45.814, E3 +61457.421}
SPL {X  -162.820, Y  +641.345, Z    +0.000, E1   +63.138, E3 +61457.468}
SPL {X  -162.820, Y  +620.039, Z    +0.000, E1   +75.979, E3 +61456.078}
SPL {X  -162.820, Y  +571.094, Z    +0.000, E1   +77.089, E3 +61471.256}
SPL {X  -158.110, Y  +341.619, Z    +0.000, E1   +77.339, E3 +61552.906}
SPL {X  -156.597, Y  +335.917, Z    +0.000, E1   +75.680, E3 +61574.749}
SPL {X  -152.710, Y  +324.020, Z    +0.000, E1   +75.365, E3 +61584.231}
SPL {X  -139.497, Y  +296.529, Z    +0.000, E1   +77.231, E3 +61577.803}
ENDSPLINE

SPLINE
SPL {X  -139.792, Y  +297.022, Z    +0.000, E1   +76.273, E3 +61586.498}
ENDSPLINE

SPLINE
SPL {X  -138.933, Y  +295.600, Z    +0.000, E1   +75.173, E3 +61596.981}
SPL {X  -137.186, Y  +292.805, Z    +0.000, E1   +73.993, E3 +61607.571}
SPL {X  -133.270, Y  +286.961, Z    +0.000, E1   +73.739, E3 +61612.285}
SPL {X  -130.283, Y  +282.844, Z    +0.000, E1   +73.297, E3 +61617.177}
SPL {X  -127.795, Y  +279.610, Z    +0.000, E1   +72.860, E3 +61621.307}
SPL {X  -124.650, Y  +275.749, Z    +0.000, E1   +72.674, E3 +61624.225}
SPL {X  -121.687, Y  +272.322, Z    +0.000, E1   +72.100, E3 +61628.534}
SPL {X  -113.980, Y  +264.229, Z    +0.000, E1   +74.120, E3 +61624.673}
SPL {X   -56.216, Y  +227.692, Z    +0.000, E1   +56.267, E3 +61801.397}
ENDSPLINE

SPLINE
SPL {X  -126.995, Y  +278.604, Z    +0.000, E1   +59.937, E3 +61973.637}
SPL {X  -150.196, Y  +317.640, Z    +0.000, E1   +49.956, E3 +61982.092}
SPL {X  -157.261, Y  +338.316, Z    +0.000, E1   +40.017, E3 +61983.787}
SPL {X  -160.924, Y  +355.726, Z    +0.000, E1   +27.715, E3 +61984.228}
SPL {X  -162.423, Y  +369.141, Z    +0.000, E1   +15.207, E3 +61984.663}
SPL {X  -162.811, Y  +378.755, Z    +0.000, E1    +4.616, E3 +61984.578}
SPL {X  -162.820, Y  +382.684, Z    +0.000, E1    -0.227, E3 +61984.132}
SPL {X  -162.820, Y  +387.227, Z    +0.000, E1   -12.320, E3 +61983.887}
SPL {X  -162.820, Y  +392.558, Z    +0.000, E1   -27.778, E3 +61983.923}
SPL {X  -162.820, Y  +400.474, Z    +0.000, E1   -46.251, E3 +61983.787}
SPL {X  -162.820, Y  +414.510, Z    +0.000, E1   -65.115, E3 +61983.230}
SPL {X  -162.820, Y  +465.064, Z    +0.000, E1   -76.269, E3 +61993.078}
SPL {X  -157.184, Y  +715.968, Z    +0.000, E1   -76.600, E3 +62089.036}
SPL {X  -156.461, Y  +718.560, Z    +0.000, E1   -75.553, E3 +62102.455}
SPL {X  -151.911, Y  +732.096, Z    +0.000, E1   -75.235, E3 +62113.009}
SPL {X  -146.569, Y  +744.407, Z    +0.000, E1   -74.677, E3 +62124.814}
SPL {X  -142.375, Y  +752.491, Z    +0.000, E1   -74.335, E3 +62131.841}
SPL {X  -139.539, Y  +757.399, Z    +0.000, E1   -73.892, E3 +62138.039}
SPL {X  -136.017, Y  +762.997, Z    +0.000, E1   -73.579, E3 +62143.221}
SPL {X  -133.089, Y  +767.296, Z    +0.000, E1   -73.251, E3 +62147.679}
SPL {X  -129.985, Y  +771.553, Z    +0.000, E1   -72.801, E3 +62152.673}
SPL {X  -126.581, Y  +775.909, Z    +0.000, E1   -72.426, E3 +62156.984}
SPL {X  -123.329, Y  +779.803, Z    +0.000, E1   -71.936, E3 +62161.366}
SPL {X  -119.291, Y  +784.315, Z    +0.000, E1   -72.148, E3 +62162.778}
SPL {X   -57.587, Y  +825.796, Z    +0.000, E1   -56.753, E3 +62316.540}
ENDSPLINE

SPLINE
SPL {X  -124.075, Y  +778.932, Z    +0.000, E1   -61.393, E3 +62510.169}
SPL {X  -150.653, Y  +735.257, Z    +0.000, E1   -50.160, E3 +62517.848}
SPL {X  -159.377, Y  +706.804, Z    +0.000, E1   -34.828, E3 +62519.492}
SPL {X  -162.134, Y  +688.425, Z    +0.000, E1   -19.100, E3 +62519.429}
SPL {X  -162.803, Y  +675.871, Z    +0.000, E1    -5.469, E3 +62519.613}
SPL {X  -162.820, Y  +671.500, Z    +0.000, E1    +0.000, E3 +62519.181}
SPL {X  -162.820, Y  +669.743, Z    +0.000, E1    +4.352, E3 +62518.976}
SPL {X  -162.820, Y  +665.917, Z    +0.000, E1   +15.272, E3 +62518.971}
SPL {X  -162.820, Y  +661.245, Z    +0.000, E1   +28.879, E3 +62518.812}
SPL {X  -162.820, Y  +654.015, Z    +0.000, E1   +45.814, E3 +62518.959}
SPL {X  -162.820, Y  +641.345, Z    +0.000, E1   +63.138, E3 +62519.006}
SPL {X  -162.820, Y  +620.039, Z    +0.000, E1   +75.979, E3 +62517.616}
SPL {X  -162.820, Y  +571.094, Z    +0.000, E1   +77.089, E3 +62532.795}
SPL {X  -157.487, Y  +339.169, Z    +0.000, E1   +76.425, E3 +62625.898}
SPL {X  -156.386, Y  +335.181, Z    +0.000, E1   +75.555, E3 +62637.959}
SPL {X  -152.710, Y  +324.020, Z    +0.000, E1   +75.365, E3 +62645.770}
SPL {X  -139.497, Y  +296.529, Z    +0.000, E1   +77.231, E3 +62639.341}
ENDSPLINE

SPLINE
SPL {X  -139.792, Y  +297.022, Z    +0.000, E1   +76.273, E3 +62648.037}
ENDSPLINE

SPLINE
SPL {X  -138.933, Y  +295.600, Z    +0.000, E1   +75.173, E3 +62658.519}
SPL {X  -137.186, Y  +292.805, Z    +0.000, E1   +73.993, E3 +62669.110}
SPL {X  -133.270, Y  +286.961, Z    +0.000, E1   +73.739, E3 +62673.823}
SPL {X  -130.283, Y  +282.844, Z    +0.000, E1   +73.297, E3 +62678.715}
SPL {X  -127.795, Y  +279.610, Z    +0.000, E1   +72.860, E3 +62682.845}
SPL {X  -124.650, Y  +275.749, Z    +0.000, E1   +72.674, E3 +62685.764}
SPL {X  -121.687, Y  +272.322, Z    +0.000, E1   +72.100, E3 +62690.073}
SPL {X  -113.980, Y  +264.229, Z    +0.000, E1   +74.120, E3 +62686.211}
SPL {X   -56.216, Y  +227.692, Z    +0.000, E1   +56.267, E3 +62862.935}
ENDSPLINE

SPLINE
SPL {X  -126.995, Y  +278.604, Z    +0.000, E1   +59.937, E3 +63035.175}
SPL {X  -150.196, Y  +317.640, Z    +0.000, E1   +49.956, E3 +63043.630}
SPL {X  -157.261, Y  +338.316, Z    +0.000, E1   +40.017, E3 +63045.326}
SPL {X  -160.924, Y  +355.726, Z    +0.000, E1   +27.715, E3 +63045.766}
SPL {X  -162.423, Y  +369.141, Z    +0.000, E1   +15.207, E3 +63046.202}
SPL {X  -162.811, Y  +378.755, Z    +0.000, E1    +4.616, E3 +63046.116}
SPL {X  -162.820, Y  +382.684, Z    +0.000, E1    -0.227, E3 +63045.671}
SPL {X  -162.820, Y  +387.227, Z    +0.000, E1   -12.320, E3 +63045.426}
SPL {X  -162.820, Y  +392.558, Z    +0.000, E1   -27.778, E3 +63045.462}
SPL {X  -162.820, Y  +400.474, Z    +0.000, E1   -46.251, E3 +63045.325}
SPL {X  -162.820, Y  +414.510, Z    +0.000, E1   -65.115, E3 +63044.769}
SPL {X  -162.820, Y  +465.064, Z    +0.000, E1   -76.269, E3 +63054.617}
SPL {X  -157.184, Y  +715.968, Z    +0.000, E1   -76.600, E3 +63150.574}
SPL {X  -156.461, Y  +718.560, Z    +0.000, E1   -75.553, E3 +63163.994}
SPL {X  -151.911, Y  +732.096, Z    +0.000, E1   -75.235, E3 +63174.548}
SPL {X  -146.569, Y  +744.407, Z    +0.000, E1   -74.677, E3 +63186.352}
SPL {X  -142.375, Y  +752.491, Z    +0.000, E1   -74.335, E3 +63193.379}
SPL {X  -139.539, Y  +757.399, Z    +0.000, E1   -73.892, E3 +63199.577}
SPL {X  -136.017, Y  +762.997, Z    +0.000, E1   -73.579, E3 +63204.759}
SPL {X  -133.089, Y  +767.296, Z    +0.000, E1   -73.251, E3 +63209.218}
SPL {X  -129.985, Y  +771.553, Z    +0.000, E1   -72.801, E3 +63214.211}
SPL {X  -126.581, Y  +775.909, Z    +0.000, E1   -72.426, E3 +63218.522}
SPL {X  -123.329, Y  +779.803, Z    +0.000, E1   -71.936, E3 +63222.904}
SPL {X  -119.291, Y  +784.315, Z    +0.000, E1   -72.148, E3 +63224.316}
SPL {X   -57.587, Y  +825.796, Z    +0.000, E1   -56.753, E3 +63378.079}
ENDSPLINE

SPLINE
SPL {X  -124.075, Y  +778.932, Z    +0.000, E1   -61.393, E3 +63571.708}
SPL {X  -150.653, Y  +735.257, Z    +0.000, E1   -50.160, E3 +63579.387}
SPL {X  -159.377, Y  +706.804, Z    +0.000, E1   -34.828, E3 +63581.030}
SPL {X  -162.134, Y  +688.425, Z    +0.000, E1   -19.100, E3 +63580.967}
SPL {X  -162.803, Y  +675.871, Z    +0.000, E1    -5.469, E3 +63581.151}
SPL {X  -162.820, Y  +671.500, Z    +0.000, E1    +0.000, E3 +63580.719}
SPL {X  -162.820, Y  +669.743, Z    +0.000, E1    +4.352, E3 +63580.515}
SPL {X  -162.820, Y  +665.917, Z    +0.000, E1   +15.272, E3 +63580.509}
SPL {X  -162.820, Y  +661.245, Z    +0.000, E1   +28.879, E3 +63580.350}
SPL {X  -162.820, Y  +654.015, Z    +0.000, E1   +45.814, E3 +63580.498}
SPL {X  -162.820, Y  +641.345, Z    +0.000, E1   +63.138, E3 +63580.545}
SPL {X  -162.820, Y  +620.039, Z    +0.000, E1   +75.979, E3 +63579.154}
SPL {X  -162.820, Y  +571.094, Z    +0.000, E1   +77.089, E3 +63594.333}
SPL {X  -157.487, Y  +339.169, Z    +0.000, E1   +76.425, E3 +63687.437}
SPL {X  -156.386, Y  +335.181, Z    +0.000, E1   +75.555, E3 +63699.498}
SPL {X  -152.710, Y  +324.020, Z    +0.000, E1   +75.365, E3 +63707.308}
SPL {X  -139.497, Y  +296.529, Z    +0.000, E1   +77.231, E3 +63700.880}
ENDSPLINE

SPLINE
SPL {X  -139.792, Y  +297.022, Z    +0.000, E1   +76.273, E3 +63709.575}
ENDSPLINE

SPLINE
SPL {X  -138.933, Y  +295.600, Z    +0.000, E1   +75.173, E3 +63720.058}
SPL {X  -137.186, Y  +292.805, Z    +0.000, E1   +73.993, E3 +63730.648}
SPL {X  -133.270, Y  +286.961, Z    +0.000, E1   +73.739, E3 +63735.362}
SPL {X  -130.283, Y  +282.844, Z    +0.000, E1   +73.297, E3 +63740.253}
SPL {X  -127.795, Y  +279.610, Z    +0.000, E1   +72.860, E3 +63744.384}
SPL {X  -124.650, Y  +275.749, Z    +0.000, E1   +72.674, E3 +63747.302}
SPL {X  -121.687, Y  +272.322, Z    +0.000, E1   +72.100, E3 +63751.611}
SPL {X  -113.980, Y  +264.229, Z    +0.000, E1   +74.120, E3 +63747.750}
SPL {X   -56.216, Y  +227.692, Z    +0.000, E1   +56.267, E3 +63924.474}
ENDSPLINE

SPLINE
SPL {X  -126.995, Y  +278.604, Z    +0.000, E1   +59.937, E3 +64096.714}
SPL {X  -150.196, Y  +317.640, Z    +0.000, E1   +49.956, E3 +64105.169}
SPL {X  -157.261, Y  +338.316, Z    +0.000, E1   +40.017, E3 +64106.864}
SPL {X  -160.924, Y  +355.726, Z    +0.000, E1   +27.715, E3 +64107.305}
SPL {X  -162.423, Y  +369.141, Z    +0.000, E1   +15.207, E3 +64107.740}
SPL {X  -162.811, Y  +378.755, Z    +0.000, E1    +4.616, E3 +64107.655}
SPL {X  -162.820, Y  +382.684, Z    +0.000, E1    -0.227, E3 +64107.209}
SPL {X  -162.820, Y  +387.227, Z    +0.000, E1   -12.320, E3 +64106.964}
SPL {X  -162.820, Y  +392.558, Z    +0.000, E1   -27.778, E3 +64107.000}
SPL {X  -162.820, Y  +400.474, Z    +0.000, E1   -46.251, E3 +64106.864}
SPL {X  -162.820, Y  +414.510, Z    +0.000, E1   -65.115, E3 +64106.307}
SPL {X  -162.820, Y  +465.064, Z    +0.000, E1   -76.269, E3 +64116.155}
SPL {X  -157.184, Y  +715.968, Z    +0.000, E1   -76.600, E3 +64212.112}
SPL {X  -156.461, Y  +718.560, Z    +0.000, E1   -75.553, E3 +64225.532}
SPL {X  -153.015, Y  +729.150, Z    +0.000, E1   -75.312, E3 +64233.621}
SPL {X  -149.053, Y  +739.025, Z    +0.000, E1   -74.952, E3 +64242.417}
SPL {X  -145.525, Y  +746.527, Z    +0.000, E1   -74.526, E3 +64250.210}
SPL {X  -142.375, Y  +752.491, Z    +0.000, E1   -74.335, E3 +64254.918}
SPL {X  -139.539, Y  +757.399, Z    +0.000, E1   -73.892, E3 +64261.116}
SPL {X  -136.017, Y  +762.997, Z    +0.000, E1   -73.579, E3 +64266.298}
SPL {X  -133.089, Y  +767.296, Z    +0.000, E1   -73.251, E3 +64270.756}
SPL {X  -129.985, Y  +771.553, Z    +0.000, E1   -72.801, E3 +64275.750}
SPL {X  -126.581, Y  +775.909, Z    +0.000, E1   -72.426, E3 +64280.061}
SPL {X  -123.329, Y  +779.803, Z    +0.000, E1   -71.936, E3 +64284.443}
SPL {X  -119.291, Y  +784.315, Z    +0.000, E1   -72.148, E3 +64285.855}
SPL {X   -57.587, Y  +825.796, Z    +0.000, E1   -56.753, E3 +64439.617}
ENDSPLINE

SPLINE
SPL {X  -124.075, Y  +778.932, Z    +0.000, E1   -61.393, E3 +64633.246}
SPL {X  -150.653, Y  +735.257, Z    +0.000, E1   -50.160, E3 +64640.925}
SPL {X  -159.377, Y  +706.804, Z    +0.000, E1   -34.828, E3 +64642.569}
SPL {X  -162.134, Y  +688.425, Z    +0.000, E1   -19.100, E3 +64642.506}
SPL {X  -162.803, Y  +675.871, Z    +0.000, E1    -5.469, E3 +64642.690}
SPL {X  -162.820, Y  +671.500, Z    +0.000, E1    +0.000, E3 +64642.258}
SPL {X  -162.820, Y  +669.743, Z    +0.000, E1    +4.352, E3 +64642.053}
SPL {X  -162.820, Y  +665.917, Z    +0.000, E1   +15.272, E3 +64642.048}
SPL {X  -162.820, Y  +659.880, Z    +0.000, E1   +32.256, E3 +64641.959}
SPL {X  -162.820, Y  +652.069, Z    +0.000, E1   +49.663, E3 +64641.985}
SPL {X  -162.820, Y  +641.345, Z    +0.000, E1   +63.138, E3 +64642.083}
SPL {X  -162.820, Y  +620.039, Z    +0.000, E1   +75.979, E3 +64640.693}
SPL {X  -162.820, Y  +571.094, Z    +0.000, E1   +77.089, E3 +64655.872}
SPL {X  -157.487, Y  +339.169, Z    +0.000, E1   +76.425, E3 +64748.975}
SPL {X  -156.386, Y  +335.181, Z    +0.000, E1   +75.555, E3 +64761.036}
SPL {X  -152.710, Y  +324.020, Z    +0.000, E1   +75.365, E3 +64768.847}
SPL {X  -139.497, Y  +296.529, Z    +0.000, E1   +77.231, E3 +64762.418}
ENDSPLINE

SPLINE
SPL {X  -139.520, Y  +296.568, Z    +0.000, E1   +75.884, E3 +64775.066}
ENDSPLINE

SPLINE
SPL {X  -138.554, Y  +294.984, Z    +0.000, E1   +74.772, E3 +64784.947}
SPL {X  -137.186, Y  +292.805, Z    +0.000, E1   +73.993, E3 +64792.187}
SPL {X  -133.270, Y  +286.961, Z    +0.000, E1   +73.739, E3 +64796.900}
SPL {X  -129.057, Y  +281.230, Z    +0.000, E1   +73.118, E3 +64803.808}
SPL {X  -123.859, Y  +274.815, Z    +0.000, E1   +72.511, E3 +64810.192}
SPL {X  -121.018, Y  +271.573, Z    +0.000, E1   +72.049, E3 +64813.710}
SPL {X  -113.980, Y  +264.229, Z    +0.000, E1   +74.120, E3 +64809.288}
SPL {X   -56.216, Y  +227.692, Z    +0.000, E1   +56.267, E3 +64986.012}
ENDSPLINE

SPLINE
SPL {X  -126.995, Y  +278.604, Z    +0.000, E1   +59.937, E3 +65158.252}
SPL {X  -150.196, Y  +317.640, Z    +0.000, E1   +49.956, E3 +65166.707}
SPL {X  -157.261, Y  +338.316, Z    +0.000, E1   +40.017, E3 +65168.402}
SPL {X  -160.924, Y  +355.726, Z    +0.000, E1   +27.715, E3 +65168.843}
SPL {X  -162.423, Y  +369.141, Z    +0.000, E1   +15.207, E3 +65169.279}
SPL {X  -162.811, Y  +378.755, Z    +0.000, E1    +4.616, E3 +65169.193}
SPL {X  -162.820, Y  +382.684, Z    +0.000, E1    -0.227, E3 +65168.748}
SPL {X  -162.820, Y  +385.721, Z    +0.000, E1    -8.371, E3 +65168.563}
SPL {X  -162.820, Y  +388.532, Z    +0.000, E1   -16.412, E3 +65168.450}
SPL {X  -162.820, Y  +392.558, Z    +0.000, E1   -27.778, E3 +65168.539}
SPL {X  -162.820, Y  +400.474, Z    +0.000, E1   -46.251, E3 +65168.402}
SPL {X  -162.820, Y  +414.510, Z    +0.000, E1   -65.115, E3 +65167.845}
SPL {X  -162.820, Y  +465.064, Z    +0.000, E1   -76.269, E3 +65177.693}
SPL {X  -157.184, Y  +715.968, Z    +0.000, E1   -76.600, E3 +65273.651}
SPL {X  -156.461, Y  +718.560, Z    +0.000, E1   -75.553, E3 +65287.071}
SPL {X  -151.911, Y  +732.096, Z    +0.000, E1   -75.235, E3 +65297.625}
SPL {X  -146.569, Y  +744.407, Z    +0.000, E1   -74.677, E3 +65309.429}
SPL {X  -142.375, Y  +752.491, Z    +0.000, E1   -74.335, E3 +65316.456}
SPL {X  -139.539, Y  +757.399, Z    +0.000, E1   -73.892, E3 +65322.654}
SPL {X  -136.017, Y  +762.997, Z    +0.000, E1   -73.579, E3 +65327.836}
SPL {X  -133.089, Y  +767.296, Z    +0.000, E1   -73.251, E3 +65332.294}
SPL {X  -129.985, Y  +771.553, Z    +0.000, E1   -72.801, E3 +65337.288}
SPL {X  -126.581, Y  +775.909, Z    +0.000, E1   -72.426, E3 +65341.599}
SPL {X  -123.329, Y  +779.803, Z    +0.000, E1   -71.936, E3 +65345.981}
SPL {X  -119.291, Y  +784.315, Z    +0.000, E1   -72.148, E3 +65347.393}
SPL {X   -57.587, Y  +825.796, Z    +0.000, E1   -56.753, E3 +65501.156}
ENDSPLINE

SPLINE
SPL {X  -124.075, Y  +778.932, Z    +0.000, E1   -61.393, E3 +65694.785}
SPL {X  -150.653, Y  +735.257, Z    +0.000, E1   -50.160, E3 +65702.464}
SPL {X  -159.377, Y  +706.804, Z    +0.000, E1   -34.828, E3 +65704.107}
SPL {X  -162.134, Y  +688.425, Z    +0.000, E1   -19.100, E3 +65704.044}
SPL {X  -162.803, Y  +675.871, Z    +0.000, E1    -5.469, E3 +65704.228}
SPL {X  -162.820, Y  +671.500, Z    +0.000, E1    +0.000, E3 +65703.796}
SPL {X  -162.820, Y  +669.743, Z    +0.000, E1    +4.352, E3 +65703.592}
SPL {X  -162.820, Y  +665.917, Z    +0.000, E1   +15.272, E3 +65703.586}
SPL {X  -162.820, Y  +661.245, Z    +0.000, E1   +28.879, E3 +65703.427}
SPL {X  -162.820, Y  +654.015, Z    +0.000, E1   +45.814, E3 +65703.574}
SPL {X  -162.820, Y  +641.345, Z    +0.000, E1   +63.138, E3 +65703.622}
SPL {X  -162.820, Y  +620.039, Z    +0.000, E1   +75.979, E3 +65702.231}
SPL {X  -162.820, Y  +571.094, Z    +0.000, E1   +77.089, E3 +65717.410}
SPL {X  -158.110, Y  +341.619, Z    +0.000, E1   +77.339, E3 +65799.060}
SPL {X  -156.597, Y  +335.917, Z    +0.000, E1   +75.680, E3 +65820.903}
SPL {X  -152.710, Y  +324.020, Z    +0.000, E1   +75.365, E3 +65830.385}
SPL {X  -139.497, Y  +296.529, Z    +0.000, E1   +77.231, E3 +65823.957}
ENDSPLINE

SPLINE
SPL {X  -139.792, Y  +297.022, Z    +0.000, E1   +76.273, E3 +65832.652}
ENDSPLINE

SPLINE
SPL {X  -138.933, Y  +295.600, Z    +0.000, E1   +75.173, E3 +65843.135}
SPL {X  -137.186, Y  +292.805, Z    +0.000, E1   +73.993, E3 +65853.725}
SPL {X  -133.270, Y  +286.961, Z    +0.000, E1   +73.739, E3 +65858.438}
SPL {X  -130.283, Y  +282.844, Z    +0.000, E1   +73.297, E3 +65863.330}
SPL {X  -127.795, Y  +279.610, Z    +0.000, E1   +72.860, E3 +65867.461}
SPL {X  -124.650, Y  +275.749, Z    +0.000, E1   +72.674, E3 +65870.379}
SPL {X  -121.687, Y  +272.322, Z    +0.000, E1   +72.100, E3 +65874.688}
SPL {X  -113.980, Y  +264.229, Z    +0.000, E1   +74.120, E3 +65870.826}
SPL {X   -56.216, Y  +227.692, Z    +0.000, E1   +56.267, E3 +66047.550}
ENDSPLINE

SPLINE
SPL {X  -126.995, Y  +278.604, Z    +0.000, E1   +59.937, E3 +66219.791}
SPL {X  -150.196, Y  +317.640, Z    +0.000, E1   +49.956, E3 +66228.246}
SPL {X  -157.261, Y  +338.316, Z    +0.000, E1   +40.017, E3 +66229.941}
SPL {X  -160.924, Y  +355.726, Z    +0.000, E1   +27.715, E3 +66230.382}
SPL {X  -162.423, Y  +369.141, Z    +0.000, E1   +15.207, E3 +66230.817}
SPL {X  -162.811, Y  +378.755, Z    +0.000, E1    +4.616, E3 +66230.732}
SPL {X  -162.820, Y  +382.684, Z    +0.000, E1    -0.227, E3 +66230.286}
SPL {X  -162.820, Y  +385.721, Z    +0.000, E1    -8.371, E3 +66230.102}
SPL {X  -162.820, Y  +388.532, Z    +0.000, E1   -16.412, E3 +66229.988}
SPL {X  -162.820, Y  +392.558, Z    +0.000, E1   -27.778, E3 +66230.077}
SPL {X  -162.820, Y  +400.474, Z    +0.000, E1   -46.251, E3 +66229.941}
SPL {X  -162.820, Y  +414.510, Z    +0.000, E1   -65.115, E3 +66229.384}
SPL {X  -162.820, Y  +465.064, Z    +0.000, E1   -76.269, E3 +66239.232}
SPL {X  -157.184, Y  +715.968, Z    +0.000, E1   -76.600, E3 +66335.189}
SPL {X  -156.461, Y  +718.560, Z    +0.000, E1   -75.553, E3 +66348.609}
SPL {X  -151.911, Y  +732.096, Z    +0.000, E1   -75.235, E3 +66359.163}
SPL {X  -146.569, Y  +744.407, Z    +0.000, E1   -74.677, E3 +66370.967}
SPL {X  -142.375, Y  +752.491, Z    +0.000, E1   -74.335, E3 +66377.995}
SPL {X  -139.539, Y  +757.399, Z    +0.000, E1   -73.892, E3 +66384.192}
SPL {X  -136.017, Y  +762.997, Z    +0.000, E1   -73.579, E3 +66389.375}
SPL {X  -133.089, Y  +767.296, Z    +0.000, E1   -73.251, E3 +66393.833}
SPL {X  -129.985, Y  +771.553, Z    +0.000, E1   -72.801, E3 +66398.827}
SPL {X  -126.581, Y  +775.909, Z    +0.000, E1   -72.426, E3 +66403.138}
SPL {X  -122.528, Y  +780.725, Z    +0.000, E1   -71.905, E3 +66408.158}
SPL {X  -116.189, Y  +787.563, Z    +0.000, E1   -72.978, E3 +66407.442}
SPL {X   -57.587, Y  +825.796, Z    +0.000, E1   -56.753, E3 +66562.694}
ENDSPLINE

SPLINE
SPL {X  -124.075, Y  +778.932, Z    +0.000, E1   -61.393, E3 +66756.323}
SPL {X  -147.028, Y  +743.450, Z    +0.000, E1   -53.078, E3 +66763.060}
SPL {X  -152.552, Y  +730.406, Z    +0.000, E1   -48.136, E3 +66764.478}
SPL {X  -159.377, Y  +706.804, Z    +0.000, E1   -34.828, E3 +66765.646}
SPL {X  -162.134, Y  +688.425, Z    +0.000, E1   -19.100, E3 +66765.583}
SPL {X  -162.803, Y  +675.871, Z    +0.000, E1    -5.469, E3 +66765.766}
SPL {X  -162.820, Y  +671.500, Z    +0.000, E1    +0.000, E3 +66765.335}
SPL {X  -162.820, Y  +669.743, Z    +0.000, E1    +4.352, E3 +66765.130}
SPL {X  -162.820, Y  +665.917, Z    +0.000, E1   +15.272, E3 +66765.125}
SPL {X  -162.820, Y  +661.245, Z    +0.000, E1   +28.879, E3 +66764.966}
SPL {X  -162.820, Y  +654.015, Z    +0.000, E1   +45.814, E3 +66765.113}
SPL {X  -162.820, Y  +641.345, Z    +0.000, E1   +63.138, E3 +66765.160}
SPL {X  -162.820, Y  +620.039, Z    +0.000, E1   +75.979, E3 +66763.770}
SPL {X  -162.820, Y  +571.094, Z    +0.000, E1   +77.089, E3 +66778.948}
SPL {X  -157.487, Y  +339.169, Z    +0.000, E1   +76.425, E3 +66872.052}
SPL {X  -156.386, Y  +335.181, Z    +0.000, E1   +75.555, E3 +66884.113}
SPL {X  -152.710, Y  +324.020, Z    +0.000, E1   +75.365, E3 +66891.924}
SPL {X  -139.497, Y  +296.529, Z    +0.000, E1   +77.231, E3 +66885.495}
ENDSPLINE

SPLINE
SPL {X  -139.520, Y  +296.568, Z    +0.000, E1   +75.884, E3 +66898.143}
ENDSPLINE

SPLINE
SPL {X  -138.554, Y  +294.984, Z    +0.000, E1   +74.772, E3 +66908.024}
SPL {X  -137.186, Y  +292.805, Z    +0.000, E1   +73.993, E3 +66915.264}
SPL {X  -133.270, Y  +286.961, Z    +0.000, E1   +73.739, E3 +66919.977}
SPL {X  -129.057, Y  +281.230, Z    +0.000, E1   +73.118, E3 +66926.885}
SPL {X  -124.650, Y  +275.749, Z    +0.000, E1   +72.674, E3 +66931.917}
SPL {X  -121.687, Y  +272.322, Z    +0.000, E1   +72.100, E3 +66936.227}
SPL {X  -113.980, Y  +264.229, Z    +0.000, E1   +74.120, E3 +66932.365}
SPL {X   -56.216, Y  +227.692, Z    +0.000, E1   +56.267, E3 +67109.089}
ENDSPLINE

SPLINE
SPL {X  -126.995, Y  +278.604, Z    +0.000, E1   +59.937, E3 +67281.329}
SPL {X  -150.196, Y  +317.640, Z    +0.000, E1   +49.956, E3 +67289.784}
SPL {X  -157.261, Y  +338.316, Z    +0.000, E1   +40.017, E3 +67291.479}
SPL {X  -160.924, Y  +355.726, Z    +0.000, E1   +27.715, E3 +67291.920}
SPL {X  -162.423, Y  +369.141, Z    +0.000, E1   +15.207, E3 +67292.356}
SPL {X  -162.811, Y  +378.755, Z    +0.000, E1    +4.616, E3 +67292.270}
SPL {X  -162.820, Y  +382.684, Z    +0.000, E1    -0.227, E3 +67291.825}
SPL {X  -162.820, Y  +387.227, Z    +0.000, E1   -12.320, E3 +67291.579}
SPL {X  -162.820, Y  +392.558, Z    +0.000, E1   -27.778, E3 +67291.616}
SPL {X  -162.820, Y  +400.474, Z    +0.000, E1   -46.251, E3 +67291.479}
SPL {X  -162.820, Y  +414.510, Z    +0.000, E1   -65.115, E3 +67290.922}
SPL {X  -162.820, Y  +465.064, Z    +0.000, E1   -76.269, E3 +67300.770}
SPL {X  -157.184, Y  +715.968, Z    +0.000, E1   -76.600, E3 +67396.728}
SPL {X  -156.461, Y  +718.560, Z    +0.000, E1   -75.553, E3 +67410.148}
SPL {X  -151.911, Y  +732.096, Z    +0.000, E1   -75.235, E3 +67420.702}
SPL {X  -146.569, Y  +744.407, Z    +0.000, E1   -74.677, E3 +67432.506}
SPL {X  -142.375, Y  +752.491, Z    +0.000, E1   -74.335, E3 +67439.533}
SPL {X  -139.539, Y  +757.399, Z    +0.000, E1   -73.892, E3 +67445.731}
SPL {X  -136.017, Y  +762.997, Z    +0.000, E1   -73.579, E3 +67450.913}
SPL {X  -133.089, Y  +767.296, Z    +0.000, E1   -73.251, E3 +67455.371}
SPL {X  -129.985, Y  +771.553, Z    +0.000, E1   -72.801, E3 +67460.365}
SPL {X  -126.581, Y  +775.909, Z    +0.000, E1   -72.426, E3 +67464.676}
SPL {X  -122.528, Y  +780.725, Z    +0.000, E1   -71.905, E3 +67469.696}
SPL {X  -116.189, Y  +787.563, Z    +0.000, E1   -72.978, E3 +67468.981}
SPL {X   -57.587, Y  +825.796, Z    +0.000, E1   -56.753, E3 +67624.233}
ENDSPLINE

SPLINE
SPL {X  -124.075, Y  +778.932, Z    +0.000, E1   -61.393, E3 +67817.862}
SPL {X  -150.653, Y  +735.257, Z    +0.000, E1   -50.160, E3 +67825.541}
SPL {X  -159.377, Y  +706.804, Z    +0.000, E1   -34.828, E3 +67827.184}
SPL {X  -162.134, Y  +688.425, Z    +0.000, E1   -19.100, E3 +67827.121}
SPL {X  -162.734, Y  +678.779, Z    +0.000, E1    -8.745, E3 +67827.260}
SPL {X  -162.820, Y  +671.589, Z    +0.000, E1    -0.221, E3 +67826.894}
SPL {X  -162.820, Y  +669.743, Z    +0.000, E1    +4.352, E3 +67826.669}
SPL {X  -162.820, Y  +665.917, Z    +0.000, E1   +15.272, E3 +67826.663}
SPL {X  -162.820, Y  +661.245, Z    +0.000, E1   +28.879, E3 +67826.504}
SPL {X  -162.820, Y  +654.015, Z    +0.000, E1   +45.814, E3 +67826.651}
SPL {X  -162.820, Y  +641.345, Z    +0.000, E1   +63.138, E3 +67826.698}
SPL {X  -162.820, Y  +620.039, Z    +0.000, E1   +75.979, E3 +67825.308}
SPL {X  -162.820, Y  +571.094, Z    +0.000, E1   +77.089, E3 +67840.487}
SPL {X  -157.487, Y  +339.169, Z    +0.000, E1   +76.425, E3 +67933.591}
SPL {X  -156.386, Y  +335.181, Z    +0.000, E1   +75.555, E3 +67945.652}
SPL {X  -152.710, Y  +324.020, Z    +0.000, E1   +75.365, E3 +67953.462}
SPL {X  -139.497, Y  +296.529, Z    +0.000, E1   +77.231, E3 +67947.034}
ENDSPLINE

SPLINE
SPL {X  -139.520, Y  +296.568, Z    +0.000, E1   +75.884, E3 +67959.681}
ENDSPLINE

SPLINE
SPL {X  -138.554, Y  +294.984, Z    +0.000, E1   +74.772, E3 +67969.562}
SPL {X  -137.186, Y  +292.805, Z    +0.000, E1   +73.993, E3 +67976.802}
SPL {X  -133.270, Y  +286.961, Z    +0.000, E1   +73.739, E3 +67981.515}
SPL {X  -129.057, Y  +281.230, Z    +0.000, E1   +73.118, E3 +67988.423}
SPL {X  -123.859, Y  +274.815, Z    +0.000, E1   +72.511, E3 +67994.808}
SPL {X  -121.018, Y  +271.573, Z    +0.000, E1   +72.049, E3 +67998.325}
SPL {X  -113.980, Y  +264.229, Z    +0.000, E1   +74.120, E3 +67993.903}
SPL {X   -56.216, Y  +227.692, Z    +0.000, E1   +56.267, E3 +68170.627}
ENDSPLINE

SPLINE
SPL {X  -126.995, Y  +278.604, Z    +0.000, E1   +59.937, E3 +68342.868}
SPL {X  -150.196, Y  +317.640, Z    +0.000, E1   +49.956, E3 +68351.323}
SPL {X  -157.261, Y  +338.316, Z    +0.000, E1   +40.017, E3 +68353.018}
SPL {X  -160.924, Y  +355.726, Z    +0.000, E1   +27.715, E3 +68353.459}
SPL {X  -162.423, Y  +369.141, Z    +0.000, E1   +15.207, E3 +68353.894}
SPL {X  -162.811, Y  +378.755, Z    +0.000, E1    +4.616, E3 +68353.808}
SPL {X  -162.820, Y  +382.684, Z    +0.000, E1    -0.227, E3 +68353.363}
SPL {X  -162.820, Y  +385.721, Z    +0.000, E1    -8.371, E3 +68353.179}
SPL {X  -162.820, Y  +388.532, Z    +0.000, E1   -16.412, E3 +68353.065}
SPL {X  -162.820, Y  +392.558, Z    +0.000, E1   -27.778, E3 +68353.154}
SPL {X  -162.820, Y  +400.474, Z    +0.000, E1   -46.251, E3 +68353.018}
SPL {X  -162.820, Y  +414.510, Z    +0.000, E1   -65.115, E3 +68352.461}
SPL {X  -162.820, Y  +465.064, Z    +0.000, E1   -76.269, E3 +68362.309}
SPL {X  -157.184, Y  +715.968, Z    +0.000, E1   -76.600, E3 +68458.266}
SPL {X  -156.461, Y  +718.560, Z    +0.000, E1   -75.553, E3 +68471.686}
SPL {X  -151.911, Y  +732.096, Z    +0.000, E1   -75.235, E3 +68482.240}
SPL {X  -146.569, Y  +744.407, Z    +0.000, E1   -74.677, E3 +68494.044}
SPL {X  -142.375, Y  +752.491, Z    +0.000, E1   -74.335, E3 +68501.072}
SPL {X  -139.539, Y  +757.399, Z    +0.000, E1   -73.892, E3 +68507.269}
SPL {X  -136.017, Y  +762.997, Z    +0.000, E1   -73.579, E3 +68512.452}
SPL {X  -133.089, Y  +767.296, Z    +0.000, E1   -73.251, E3 +68516.910}
SPL {X  -129.985, Y  +771.553, Z    +0.000, E1   -72.801, E3 +68521.904}
SPL {X  -126.581, Y  +775.909, Z    +0.000, E1   -72.426, E3 +68526.215}
SPL {X  -122.528, Y  +780.725, Z    +0.000, E1   -71.905, E3 +68531.235}
SPL {X  -116.189, Y  +787.563, Z    +0.000, E1   -72.978, E3 +68530.519}
SPL {X   -57.587, Y  +825.796, Z    +0.000, E1   -56.753, E3 +68685.771}
ENDSPLINE

SPLINE
SPL {X  -124.075, Y  +778.932, Z    +0.000, E1   -61.393, E3 +68879.400}
SPL {X  -147.028, Y  +743.450, Z    +0.000, E1   -53.078, E3 +68886.137}
SPL {X  -152.552, Y  +730.406, Z    +0.000, E1   -48.136, E3 +68887.555}
SPL {X  -159.377, Y  +706.804, Z    +0.000, E1   -34.828, E3 +68888.723}
SPL {X  -162.134, Y  +688.425, Z    +0.000, E1   -19.100, E3 +68888.659}
SPL {X  -162.803, Y  +675.871, Z    +0.000, E1    -5.469, E3 +68888.843}
SPL {X  -162.820, Y  +671.500, Z    +0.000, E1    +0.000, E3 +68888.411}
SPL {X  -162.820, Y  +669.743, Z    +0.000, E1    +4.352, E3 +68888.207}
SPL {X  -162.820, Y  +665.917, Z    +0.000, E1   +15.272, E3 +68888.202}
SPL {X  -162.820, Y  +661.245, Z    +0.000, E1   +28.879, E3 +68888.043}
SPL {X  -162.820, Y  +654.015, Z    +0.000, E1   +45.814, E3 +68888.190}
SPL {X  -162.820, Y  +641.345, Z    +0.000, E1   +63.138, E3 +68888.237}
SPL {X  -162.820, Y  +620.039, Z    +0.000, E1   +75.979, E3 +68886.847}
SPL {X  -162.820, Y  +571.094, Z    +0.000, E1   +77.089, E3 +68902.025}
SPL {X  -157.487, Y  +339.169, Z    +0.000, E1   +76.425, E3 +68995.129}
SPL {X  -156.386, Y  +335.181, Z    +0.000, E1   +75.555, E3 +69007.190}
SPL {X  -152.710, Y  +324.020, Z    +0.000, E1   +75.365, E3 +69015.000}
SPL {X  -139.497, Y  +296.529, Z    +0.000, E1   +77.231, E3 +69008.572}
ENDSPLINE

SPLINE
SPL {X  -139.792, Y  +297.022, Z    +0.000, E1   +76.273, E3 +69017.267}
ENDSPLINE

SPLINE
SPL {X  -139.059, Y  +295.807, Z    +0.000, E1   +75.126, E3 +69028.085}
ENDSPLINE

SPLINE
SPL {X  -141.801, Y  +300.482, Z    +0.000, E1   +72.738, E3 +69044.456}
ENDSPLINE

SPLINE
SPL {X  -138.166, Y  +294.358, Z    +0.000, E1   +72.281, E3 +69051.297}
SPL {X  -134.385, Y  +288.571, Z    +0.000, E1   +71.826, E3 +69057.561}
SPL {X  -130.773, Y  +283.501, Z    +0.000, E1   +71.398, E3 +69062.985}
SPL {X  -126.922, Y  +278.513, Z    +0.000, E1   +70.767, E3 +69069.139}
SPL {X  -123.520, Y  +274.419, Z    +0.000, E1   +70.342, E3 +69073.338}
SPL {X  -117.513, Y  +267.801, Z    +0.000, E1   +72.197, E3 +69069.687}
SPL {X   -63.140, Y  +230.421, Z    +0.000, E1   +55.875, E3 +69239.125}
ENDSPLINE

SPLINE
SPL {X  -130.329, Y  +282.905, Z    +0.000, E1   +55.659, E3 +69397.461}
SPL {X  -150.766, Y  +319.018, Z    +0.000, E1   +45.408, E3 +69405.954}
SPL {X  -157.479, Y  +339.138, Z    +0.000, E1   +35.556, E3 +69407.390}
SPL {X  -160.994, Y  +356.185, Z    +0.000, E1   +24.373, E3 +69409.435}
SPL {X  -162.352, Y  +368.168, Z    +0.000, E1   +14.282, E3 +69409.488}
SPL {X  -162.808, Y  +378.562, Z    +0.000, E1    +4.298, E3 +69409.420}
SPL {X  -162.820, Y  +382.500, Z    +0.000, E1    +0.000, E3 +69408.993}
SPL {X  -162.820, Y  +384.915, Z    +0.000, E1    -4.894, E3 +69408.706}
SPL {X  -162.820, Y  +388.986, Z    +0.000, E1   -15.047, E3 +69408.804}
SPL {X  -162.820, Y  +394.732, Z    +0.000, E1   -28.992, E3 +69408.655}
SPL {X  -162.820, Y  +403.075, Z    +0.000, E1   -46.096, E3 +69408.885}
SPL {X  -162.820, Y  +414.705, Z    +0.000, E1   -61.052, E3 +69408.331}
SPL {X  -162.820, Y  +466.149, Z    +0.000, E1   -74.732, E3 +69418.327}
SPL {X  -160.722, Y  +699.554, Z    +0.000, E1   -75.485, E3 +69515.737}
SPL {X  -159.966, Y  +703.854, Z    +0.000, E1   -74.386, E3 +69530.641}
SPL {X  -156.868, Y  +717.123, Z    +0.000, E1   -74.182, E3 +69540.319}
SPL {X  -153.226, Y  +728.564, Z    +0.000, E1   -73.755, E3 +69551.327}
SPL {X  -149.090, Y  +738.941, Z    +0.000, E1   -73.348, E3 +69560.901}
SPL {X  -145.714, Y  +746.149, Z    +0.000, E1   -72.951, E3 +69568.487}
SPL {X  -140.946, Y  +755.015, Z    +0.000, E1   -72.452, E3 +69577.590}
SPL {X  -136.902, Y  +761.638, Z    +0.000, E1   -71.857, E3 +69585.457}
SPL {X  -133.350, Y  +766.925, Z    +0.000, E1   -71.498, E3 +69590.778}
SPL {X  -129.687, Y  +771.946, Z    +0.000, E1   -71.061, E3 +69596.144}
SPL {X  -126.374, Y  +776.164, Z    +0.000, E1   -70.494, E3 +69601.397}
SPL {X  -122.717, Y  +780.508, Z    +0.000, E1   -70.361, E3 +69604.435}
SPL {X  -114.093, Y  +789.660, Z    +0.000, E1   -71.634, E3 +69604.453}
SPL {X   -61.593, Y  +824.220, Z    +0.000, E1   -55.970, E3 +69770.289}
ENDSPLINE

SPLINE
SPL {X  -131.598, Y  +769.376, Z    +0.000, E1   -56.871, E3 +69936.560}
SPL {X  -152.760, Y  +729.846, Z    +0.000, E1   -44.713, E3 +69943.613}
SPL {X  -158.868, Y  +709.157, Z    +0.000, E1   -33.466, E3 +69944.814}
SPL {X  -161.987, Y  +689.949, Z    +0.000, E1   -18.777, E3 +69945.775}
SPL {X  -162.803, Y  +675.860, Z    +0.000, E1    -4.958, E3 +69945.757}
SPL {X  -162.820, Y  +671.500, Z    +0.000, E1    +0.000, E3 +69945.293}
SPL {X  -162.820, Y  +669.410, Z    +0.000, E1    +4.515, E3 +69945.056}
SPL {X  -162.820, Y  +664.781, Z    +0.000, E1   +16.411, E3 +69945.051}
SPL {X  -162.820, Y  +659.650, Z    +0.000, E1   +29.778, E3 +69945.061}
SPL {X  -162.820, Y  +651.175, Z    +0.000, E1   +47.162, E3 +69945.211}
SPL {X  -162.820, Y  +637.134, Z    +0.000, E1   +65.232, E3 +69943.753}
SPL {X  -162.820, Y  +616.721, Z    +0.000, E1   +72.273, E3 +69947.487}
SPL {X  -162.820, Y  +577.172, Z    +0.000, E1   +75.843, E3 +69957.467}
SPL {X  -159.895, Y  +349.775, Z    +0.000, E1   +76.042, E3 +70049.133}
ENDSPLINE

SPLINE
SPL {X  -160.357, Y  +352.285, Z    +0.000, E1   +74.783, E3 +70062.071}
ENDSPLINE

SPLINE
SPL {X  -145.737, Y  +307.897, Z    +0.000, E1   +77.368, E3 +70054.646}
SPL {X  -145.329, Y  +307.084, Z    +0.000, E1   +76.571, E3 +70063.482}
ENDSPLINE

SPLINE
SPL {X  -145.355, Y  +307.136, Z    +0.000, E1   +75.607, E3 +70073.007}
ENDSPLINE

SPLINE
SPL {X  -144.515, Y  +305.495, Z    +0.000, E1   +74.543, E3 +70083.816}
SPL {X  -143.690, Y  +303.925, Z    +0.000, E1   +73.372, E3 +70094.554}
SPL {X  -141.993, Y  +300.823, Z    +0.000, E1   +72.659, E3 +70101.979}
SPL {X  -138.166, Y  +294.358, Z    +0.000, E1   +72.281, E3 +70108.440}
SPL {X  -134.385, Y  +288.571, Z    +0.000, E1   +71.826, E3 +70114.704}
SPL {X  -130.773, Y  +283.501, Z    +0.000, E1   +71.398, E3 +70120.128}
SPL {X  -126.922, Y  +278.513, Z    +0.000, E1   +70.767, E3 +70126.282}
SPL {X  -123.520, Y  +274.419, Z    +0.000, E1   +70.342, E3 +70130.481}
SPL {X  -117.513, Y  +267.801, Z    +0.000, E1   +72.197, E3 +70126.830}
SPL {X   -63.140, Y  +230.421, Z    +0.000, E1   +55.875, E3 +70296.268}
ENDSPLINE

SPLINE
SPL {X  -130.329, Y  +282.905, Z    +0.000, E1   +55.659, E3 +70454.604}
SPL {X  -154.728, Y  +329.807, Z    +0.000, E1   +40.640, E3 +70463.985}
SPL {X  -160.994, Y  +356.185, Z    +0.000, E1   +24.373, E3 +70466.578}
SPL {X  -162.637, Y  +372.778, Z    +0.000, E1   +10.098, E3 +70466.598}
SPL {X  -162.820, Y  +382.748, Z    +0.000, E1    -0.178, E3 +70466.091}
SPL {X  -162.820, Y  +387.647, Z    +0.000, E1   -11.488, E3 +70465.880}
SPL {X  -162.820, Y  +393.007, Z    +0.000, E1   -25.093, E3 +70465.838}
SPL {X  -162.820, Y  +400.636, Z    +0.000, E1   -41.711, E3 +70465.888}
SPL {X  -162.820, Y  +414.705, Z    +0.000, E1   -61.052, E3 +70465.474}
SPL {X  -162.820, Y  +466.149, Z    +0.000, E1   -74.732, E3 +70475.470}
SPL {X  -160.066, Y  +703.318, Z    +0.000, E1   -76.774, E3 +70560.318}
ENDSPLINE

SPLINE
SPL {X  -161.105, Y  +697.069, Z    +0.000, E1   -74.557, E3 +70581.932}
ENDSPLINE

SPLINE
SPL {X  -159.270, Y  +707.314, Z    +0.000, E1   -74.359, E3 +70589.956}
SPL {X  -156.868, Y  +717.123, Z    +0.000, E1   -74.182, E3 +70597.462}
SPL {X  -154.373, Y  +725.261, Z    +0.000, E1   -73.879, E3 +70605.172}
SPL {X  -152.060, Y  +731.708, Z    +0.000, E1   -73.572, E3 +70611.820}
SPL {X  -149.090, Y  +738.941, Z    +0.000, E1   -73.348, E3 +70618.043}
SPL {X  -145.714, Y  +746.149, Z    +0.000, E1   -72.951, E3 +70625.630}
SPL {X  -140.946, Y  +755.015, Z    +0.000, E1   -72.452, E3 +70634.733}
SPL {X  -136.902, Y  +761.638, Z    +0.000, E1   -71.857, E3 +70642.600}
SPL {X  -133.350, Y  +766.925, Z    +0.000, E1   -71.498, E3 +70647.920}
SPL {X  -129.687, Y  +771.946, Z    +0.000, E1   -71.061, E3 +70653.286}
SPL {X  -126.374, Y  +776.164, Z    +0.000, E1   -70.494, E3 +70658.540}
SPL {X  -122.717, Y  +780.508, Z    +0.000, E1   -70.361, E3 +70661.577}
SPL {X  -114.093, Y  +789.660, Z    +0.000, E1   -71.634, E3 +70661.596}
SPL {X   -61.795, Y  +824.138, Z    +0.000, E1   -56.629, E3 +70807.263}
ENDSPLINE

SPLINE
SPL {X  -113.687, Y  +790.058, Z    +0.000, E1   -59.721, E3 +70984.010}
SPL {X  -139.151, Y  +758.042, Z    +0.000, E1   -54.091, E3 +70995.569}
SPL {X  -152.760, Y  +729.846, Z    +0.000, E1   -44.713, E3 +71000.756}
SPL {X  -158.868, Y  +709.157, Z    +0.000, E1   -33.466, E3 +71001.957}
SPL {X  -161.987, Y  +689.949, Z    +0.000, E1   -18.777, E3 +71002.918}
SPL {X  -162.743, Y  +678.515, Z    +0.000, E1    -7.658, E3 +71002.913}
SPL {X  -162.820, Y  +671.380, Z    +0.000, E1    +0.035, E3 +71002.418}
SPL {X  -162.820, Y  +668.318, Z    +0.000, E1    +7.404, E3 +71002.155}
SPL {X  -162.820, Y  +664.781, Z    +0.000, E1   +16.411, E3 +71002.194}
SPL {X  -162.820, Y  +659.650, Z    +0.000, E1   +29.778, E3 +71002.204}
SPL {X  -162.820, Y  +651.175, Z    +0.000, E1   +47.162, E3 +71002.353}
SPL {X  -162.820, Y  +633.243, Z    +0.000, E1   +67.111, E3 +71001.608}
SPL {X  -162.820, Y  +577.172, Z    +0.000, E1   +75.843, E3 +71014.610}
SPL {X  -159.895, Y  +349.775, Z    +0.000, E1   +76.042, E3 +71106.276}
ENDSPLINE

SPLINE
SPL {X  -160.357, Y  +352.285, Z    +0.000, E1   +74.783, E3 +71119.214}
ENDSPLINE

SPLINE
SPL {X  -145.737, Y  +307.897, Z    +0.000, E1   +77.368, E3 +71111.789}
SPL {X  -145.329, Y  +307.084, Z    +0.000, E1   +76.571, E3 +71120.625}
ENDSPLINE

SPLINE
SPL {X  -145.355, Y  +307.136, Z    +0.000, E1   +75.607, E3 +71130.149}
ENDSPLINE

SPLINE
SPL {X  -144.515, Y  +305.495, Z    +0.000, E1   +74.543, E3 +71140.959}
SPL {X  -143.690, Y  +303.925, Z    +0.000, E1   +73.372, E3 +71151.697}
SPL {X  -141.993, Y  +300.823, Z    +0.000, E1   +72.659, E3 +71159.122}
SPL {X  -138.166, Y  +294.358, Z    +0.000, E1   +72.281, E3 +71165.583}
SPL {X  -134.385, Y  +288.571, Z    +0.000, E1   +71.826, E3 +71171.847}
SPL {X  -129.872, Y  +282.297, Z    +0.000, E1   +71.229, E3 +71179.017}
SPL {X  -124.448, Y  +275.510, Z    +0.000, E1   +70.509, E3 +71186.390}
SPL {X  -117.513, Y  +267.801, Z    +0.000, E1   +72.197, E3 +71183.972}
SPL {X   -63.140, Y  +230.421, Z    +0.000, E1   +55.875, E3 +71353.411}
ENDSPLINE

SPLINE
SPL {X  -130.329, Y  +282.905, Z    +0.000, E1   +55.659, E3 +71511.747}
SPL {X  -150.766, Y  +319.018, Z    +0.000, E1   +45.408, E3 +71520.240}
SPL {X  -157.479, Y  +339.138, Z    +0.000, E1   +35.556, E3 +71521.675}
SPL {X  -160.994, Y  +356.185, Z    +0.000, E1   +24.373, E3 +71523.721}
SPL {X  -162.352, Y  +368.168, Z    +0.000, E1   +14.282, E3 +71523.774}
SPL {X  -162.808, Y  +378.562, Z    +0.000, E1    +4.298, E3 +71523.706}
SPL {X  -162.820, Y  +382.500, Z    +0.000, E1    +0.000, E3 +71523.278}
SPL {X  -162.820, Y  +384.915, Z    +0.000, E1    -4.894, E3 +71522.992}
SPL {X  -162.820, Y  +388.986, Z    +0.000, E1   -15.047, E3 +71523.090}
SPL {X  -162.820, Y  +394.732, Z    +0.000, E1   -28.992, E3 +71522.941}
SPL {X  -162.820, Y  +403.075, Z    +0.000, E1   -46.096, E3 +71523.171}
SPL {X  -162.820, Y  +414.705, Z    +0.000, E1   -61.052, E3 +71522.617}
SPL {X  -162.820, Y  +466.149, Z    +0.000, E1   -74.732, E3 +71532.613}
SPL {X  -160.722, Y  +699.554, Z    +0.000, E1   -75.485, E3 +71630.023}
SPL {X  -159.966, Y  +703.854, Z    +0.000, E1   -74.386, E3 +71644.926}
SPL {X  -156.868, Y  +717.123, Z    +0.000, E1   -74.182, E3 +71654.605}
SPL {X  -153.226, Y  +728.564, Z    +0.000, E1   -73.755, E3 +71665.613}
SPL {X  -149.090, Y  +738.941, Z    +0.000, E1   -73.348, E3 +71675.186}
SPL {X  -145.714, Y  +746.149, Z    +0.000, E1   -72.951, E3 +71682.773}
SPL {X  -140.946, Y  +755.015, Z    +0.000, E1   -72.452, E3 +71691.876}
SPL {X  -136.902, Y  +761.638, Z    +0.000, E1   -71.857, E3 +71699.743}
SPL {X  -133.350, Y  +766.925, Z    +0.000, E1   -71.498, E3 +71705.063}
SPL {X  -129.687, Y  +771.946, Z    +0.000, E1   -71.061, E3 +71710.429}
SPL {X  -126.374, Y  +776.164, Z    +0.000, E1   -70.494, E3 +71715.683}
SPL {X  -122.717, Y  +780.508, Z    +0.000, E1   -70.361, E3 +71718.720}
SPL {X  -114.093, Y  +789.660, Z    +0.000, E1   -71.634, E3 +71718.738}
SPL {X   -61.795, Y  +824.138, Z    +0.000, E1   -56.629, E3 +71864.406}
ENDSPLINE

SPLINE
SPL {X  -113.687, Y  +790.058, Z    +0.000, E1   -59.721, E3 +72041.153}
SPL {X  -139.151, Y  +758.042, Z    +0.000, E1   -54.091, E3 +72052.712}
SPL {X  -152.760, Y  +729.846, Z    +0.000, E1   -44.713, E3 +72057.898}
SPL {X  -158.868, Y  +709.157, Z    +0.000, E1   -33.466, E3 +72059.099}
SPL {X  -161.987, Y  +689.949, Z    +0.000, E1   -18.777, E3 +72060.061}
SPL {X  -162.743, Y  +678.515, Z    +0.000, E1    -7.658, E3 +72060.056}
SPL {X  -162.820, Y  +671.380, Z    +0.000, E1    +0.035, E3 +72059.560}
SPL {X  -162.820, Y  +668.318, Z    +0.000, E1    +7.404, E3 +72059.298}
SPL {X  -162.820, Y  +664.781, Z    +0.000, E1   +16.411, E3 +72059.337}
SPL {X  -162.820, Y  +659.650, Z    +0.000, E1   +29.778, E3 +72059.346}
SPL {X  -162.820, Y  +651.175, Z    +0.000, E1   +47.162, E3 +72059.496}
SPL {X  -162.820, Y  +633.243, Z    +0.000, E1   +67.111, E3 +72058.751}
SPL {X  -162.820, Y  +577.172, Z    +0.000, E1   +75.843, E3 +72071.753}
SPL {X  -159.895, Y  +349.775, Z    +0.000, E1   +76.042, E3 +72163.419}
ENDSPLINE

SPLINE
SPL {X  -160.357, Y  +352.285, Z    +0.000, E1   +74.783, E3 +72176.357}
ENDSPLINE

SPLINE
SPL {X  -145.737, Y  +307.897, Z    +0.000, E1   +77.368, E3 +72168.932}
SPL {X  -145.329, Y  +307.084, Z    +0.000, E1   +76.571, E3 +72177.768}
ENDSPLINE

SPLINE
SPL {X  -145.355, Y  +307.136, Z    +0.000, E1   +75.607, E3 +72187.292}
ENDSPLINE

SPLINE
SPL {X  -144.515, Y  +305.495, Z    +0.000, E1   +74.543, E3 +72198.101}
SPL {X  -143.690, Y  +303.925, Z    +0.000, E1   +73.372, E3 +72208.840}
SPL {X  -141.993, Y  +300.823, Z    +0.000, E1   +72.659, E3 +72216.265}
SPL {X  -138.166, Y  +294.358, Z    +0.000, E1   +72.281, E3 +72222.726}
SPL {X  -134.385, Y  +288.571, Z    +0.000, E1   +71.826, E3 +72228.990}
SPL {X  -129.872, Y  +282.297, Z    +0.000, E1   +71.229, E3 +72236.160}
SPL {X  -124.448, Y  +275.510, Z    +0.000, E1   +70.509, E3 +72243.533}
SPL {X  -117.513, Y  +267.801, Z    +0.000, E1   +72.197, E3 +72241.115}
SPL {X   -63.140, Y  +230.421, Z    +0.000, E1   +55.875, E3 +72410.554}
ENDSPLINE

SPLINE
SPL {X  -130.329, Y  +282.905, Z    +0.000, E1   +55.659, E3 +72568.890}
SPL {X  -154.728, Y  +329.807, Z    +0.000, E1   +40.640, E3 +72578.271}
SPL {X  -160.994, Y  +356.185, Z    +0.000, E1   +24.373, E3 +72580.864}
SPL {X  -162.637, Y  +372.778, Z    +0.000, E1   +10.098, E3 +72580.884}
SPL {X  -162.820, Y  +382.748, Z    +0.000, E1    -0.178, E3 +72580.377}
SPL {X  -162.820, Y  +387.647, Z    +0.000, E1   -11.488, E3 +72580.166}
SPL {X  -162.820, Y  +393.007, Z    +0.000, E1   -25.093, E3 +72580.124}
SPL {X  -162.820, Y  +400.636, Z    +0.000, E1   -41.711, E3 +72580.173}
SPL {X  -162.820, Y  +414.705, Z    +0.000, E1   -61.052, E3 +72579.760}
SPL {X  -162.820, Y  +466.149, Z    +0.000, E1   -74.732, E3 +72589.756}
SPL {X  -160.722, Y  +699.554, Z    +0.000, E1   -75.485, E3 +72687.166}
SPL {X  -159.966, Y  +703.854, Z    +0.000, E1   -74.386, E3 +72702.069}
SPL {X  -156.868, Y  +717.123, Z    +0.000, E1   -74.182, E3 +72711.747}
SPL {X  -153.226, Y  +728.564, Z    +0.000, E1   -73.755, E3 +72722.756}
SPL {X  -149.090, Y  +738.941, Z    +0.000, E1   -73.348, E3 +72732.329}
SPL {X  -145.714, Y  +746.149, Z    +0.000, E1   -72.951, E3 +72739.916}
SPL {X  -140.946, Y  +755.015, Z    +0.000, E1   -72.452, E3 +72749.019}
SPL {X  -136.902, Y  +761.638, Z    +0.000, E1   -71.857, E3 +72756.886}
SPL {X  -133.350, Y  +766.925, Z    +0.000, E1   -71.498, E3 +72762.206}
SPL {X  -129.687, Y  +771.946, Z    +0.000, E1   -71.061, E3 +72767.572}
SPL {X  -126.374, Y  +776.164, Z    +0.000, E1   -70.494, E3 +72772.826}
SPL {X  -123.763, Y  +779.297, Z    +0.000, E1   -70.128, E3 +72776.201}
SPL {X  -119.350, Y  +784.252, Z    +0.000, E1   -71.016, E3 +72775.402}
SPL {X   -61.593, Y  +824.220, Z    +0.000, E1   -55.970, E3 +72941.717}
ENDSPLINE

SPLINE
SPL {X  -131.598, Y  +769.376, Z    +0.000, E1   -56.871, E3 +73107.989}
SPL {X  -152.760, Y  +729.846, Z    +0.000, E1   -44.713, E3 +73115.041}
SPL {X  -158.868, Y  +709.157, Z    +0.000, E1   -33.466, E3 +73116.242}
SPL {X  -161.987, Y  +689.949, Z    +0.000, E1   -18.777, E3 +73117.203}
SPL {X  -162.803, Y  +675.860, Z    +0.000, E1    -4.958, E3 +73117.186}
SPL {X  -162.820, Y  +671.500, Z    +0.000, E1    +0.000, E3 +73116.722}
SPL {X  -162.820, Y  +669.410, Z    +0.000, E1    +4.515, E3 +73116.484}
SPL {X  -162.820, Y  +664.781, Z    +0.000, E1   +16.411, E3 +73116.480}
SPL {X  -162.820, Y  +659.650, Z    +0.000, E1   +29.778, E3 +73116.489}
SPL {X  -162.820, Y  +654.031, Z    +0.000, E1   +42.449, E3 +73116.403}
SPL {X  -162.820, Y  +647.611, Z    +0.000, E1   +52.483, E3 +73116.933}
SPL {X  -162.820, Y  +633.243, Z    +0.000, E1   +67.111, E3 +73115.894}
SPL {X  -162.820, Y  +577.172, Z    +0.000, E1   +75.843, E3 +73128.896}
SPL {X  -159.895, Y  +349.775, Z    +0.000, E1   +76.042, E3 +73220.562}
ENDSPLINE

SPLINE
SPL {X  -160.357, Y  +352.285, Z    +0.000, E1   +74.783, E3 +73233.500}
ENDSPLINE

SPLINE
SPL {X  -145.737, Y  +307.897, Z    +0.000, E1   +77.368, E3 +73226.075}
SPL {X  -145.329, Y  +307.084, Z    +0.000, E1   +76.571, E3 +73234.911}
ENDSPLINE

SPLINE
SPL {X  -145.355, Y  +307.136, Z    +0.000, E1   +75.607, E3 +73244.435}
ENDSPLINE

SPLINE
SPL {X  -144.515, Y  +305.495, Z    +0.000, E1   +74.543, E3 +73255.244}
SPL {X  -143.690, Y  +303.925, Z    +0.000, E1   +73.372, E3 +73265.983}
SPL {X  -141.993, Y  +300.823, Z    +0.000, E1   +72.659, E3 +73273.408}
SPL {X  -138.166, Y  +294.358, Z    +0.000, E1   +72.281, E3 +73279.869}
SPL {X  -134.385, Y  +288.571, Z    +0.000, E1   +71.826, E3 +73286.132}
SPL {X  -130.773, Y  +283.501, Z    +0.000, E1   +71.398, E3 +73291.557}
SPL {X  -126.922, Y  +278.513, Z    +0.000, E1   +70.767, E3 +73297.711}
SPL {X  -123.520, Y  +274.419, Z    +0.000, E1   +70.342, E3 +73301.909}
SPL {X  -117.513, Y  +267.801, Z    +0.000, E1   +72.197, E3 +73298.258}
SPL {X   -63.140, Y  +230.421, Z    +0.000, E1   +55.875, E3 +73467.697}
ENDSPLINE

SPLINE
SPL {X  -130.329, Y  +282.905, Z    +0.000, E1   +55.659, E3 +73626.033}
SPL {X  -154.728, Y  +329.807, Z    +0.000, E1   +40.640, E3 +73635.414}
SPL {X  -160.994, Y  +356.185, Z    +0.000, E1   +24.373, E3 +73638.007}
SPL {X  -162.352, Y  +368.168, Z    +0.000, E1   +14.282, E3 +73638.059}
SPL {X  -162.808, Y  +378.562, Z    +0.000, E1    +4.298, E3 +73637.991}
SPL {X  -162.820, Y  +382.500, Z    +0.000, E1    +0.000, E3 +73637.564}
SPL {X  -162.820, Y  +384.915, Z    +0.000, E1    -4.894, E3 +73637.277}
SPL {X  -162.820, Y  +388.986, Z    +0.000, E1   -15.047, E3 +73637.375}
SPL {X  -162.820, Y  +393.007, Z    +0.000, E1   -25.093, E3 +73637.266}
SPL {X  -162.820, Y  +400.636, Z    +0.000, E1   -41.711, E3 +73637.316}
SPL {X  -162.820, Y  +414.705, Z    +0.000, E1   -61.052, E3 +73636.903}
SPL {X  -162.820, Y  +466.149, Z    +0.000, E1   -74.732, E3 +73646.899}
SPL {X  -160.722, Y  +699.554, Z    +0.000, E1   -75.485, E3 +73744.309}
SPL {X  -159.966, Y  +703.854, Z    +0.000, E1   -74.386, E3 +73759.212}
SPL {X  -156.868, Y  +717.123, Z    +0.000, E1   -74.182, E3 +73768.890}
SPL {X  -153.226, Y  +728.564, Z    +0.000, E1   -73.755, E3 +73779.898}
SPL {X  -149.090, Y  +738.941, Z    +0.000, E1   -73.348, E3 +73789.472}
SPL {X  -145.714, Y  +746.149, Z    +0.000, E1   -72.951, E3 +73797.059}
SPL {X  -140.946, Y  +755.015, Z    +0.000, E1   -72.452, E3 +73806.162}
SPL {X  -136.902, Y  +761.638, Z    +0.000, E1   -71.857, E3 +73814.028}
SPL {X  -133.350, Y  +766.925, Z    +0.000, E1   -71.498, E3 +73819.349}
SPL {X  -129.687, Y  +771.946, Z    +0.000, E1   -71.061, E3 +73824.715}
SPL {X  -126.374, Y  +776.164, Z    +0.000, E1   -70.494, E3 +73829.968}
SPL {X  -123.763, Y  +779.297, Z    +0.000, E1   -70.128, E3 +73833.344}
SPL {X  -119.350, Y  +784.252, Z    +0.000, E1   -71.016, E3 +73832.544}
SPL {X   -61.593, Y  +824.220, Z    +0.000, E1   -55.970, E3 +73998.860}
ENDSPLINE

SPLINE
SPL {X  -131.598, Y  +769.376, Z    +0.000, E1   -56.871, E3 +74165.132}
SPL {X  -152.760, Y  +729.846, Z    +0.000, E1   -44.713, E3 +74172.184}
SPL {X  -158.868, Y  +709.157, Z    +0.000, E1   -33.466, E3 +74173.385}
SPL {X  -161.987, Y  +689.949, Z    +0.000, E1   -18.777, E3 +74174.346}
SPL {X  -162.803, Y  +675.860, Z    +0.000, E1    -4.958, E3 +74174.328}
SPL {X  -162.820, Y  +671.500, Z    +0.000, E1    +0.000, E3 +74173.865}
SPL {X  -162.820, Y  +669.410, Z    +0.000, E1    +4.515, E3 +74173.627}
SPL {X  -162.820, Y  +664.781, Z    +0.000, E1   +16.411, E3 +74173.622}
SPL {X  -162.820, Y  +659.650, Z    +0.000, E1   +29.778, E3 +74173.632}
SPL {X  -162.820, Y  +654.031, Z    +0.000, E1   +42.449, E3 +74173.546}
SPL {X  -162.820, Y  +647.611, Z    +0.000, E1   +52.483, E3 +74174.076}
SPL {X  -162.820, Y  +637.134, Z    +0.000, E1   +65.232, E3 +74172.324}
SPL {X  -162.820, Y  +616.721, Z    +0.000, E1   +72.273, E3 +74176.058}
SPL {X  -162.820, Y  +577.172, Z    +0.000, E1   +75.843, E3 +74186.039}
SPL {X  -159.895, Y  +349.775, Z    +0.000, E1   +76.042, E3 +74277.705}
ENDSPLINE

SPLINE
SPL {X  -160.357, Y  +352.285, Z    +0.000, E1   +74.783, E3 +74290.642}
ENDSPLINE

SPLINE
SPL {X  -145.737, Y  +307.897, Z    +0.000, E1   +77.368, E3 +74283.218}
SPL {X  -145.122, Y  +306.676, Z    +0.000, E1   +76.360, E3 +74294.571}
ENDSPLINE

SPLINE
SPL {X  -145.186, Y  +306.802, Z    +0.000, E1   +74.850, E3 +74308.924}
ENDSPLINE

SPLINE
SPL {X  -143.742, Y  +304.025, Z    +0.000, E1   +73.644, E3 +74320.978}
SPL {X  -141.993, Y  +300.823, Z    +0.000, E1   +72.659, E3 +74330.551}
SPL {X  -138.166, Y  +294.358, Z    +0.000, E1   +72.281, E3 +74337.012}
SPL {X  -134.385, Y  +288.571, Z    +0.000, E1   +71.826, E3 +74343.275}
SPL {X  -129.872, Y  +282.297, Z    +0.000, E1   +71.229, E3 +74350.445}
SPL {X  -124.448, Y  +275.510, Z    +0.000, E1   +70.509, E3 +74357.818}
SPL {X  -117.513, Y  +267.801, Z    +0.000, E1   +72.197, E3 +74355.401}
SPL {X   -63.140, Y  +230.421, Z    +0.000, E1   +55.875, E3 +74524.840}
ENDSPLINE

SPLINE
SPL {X  -130.329, Y  +282.905, Z    +0.000, E1   +55.659, E3 +74683.176}
SPL {X  -154.728, Y  +329.807, Z    +0.000, E1   +40.640, E3 +74692.557}
SPL {X  -160.994, Y  +356.185, Z    +0.000, E1   +24.373, E3 +74695.150}
SPL {X  -162.637, Y  +372.778, Z    +0.000, E1   +10.098, E3 +74695.170}
SPL {X  -162.820, Y  +382.419, Z    +0.000, E1    +0.163, E3 +74694.730}
SPL {X  -162.820, Y  +384.915, Z    +0.000, E1    -4.894, E3 +74694.420}
SPL {X  -162.820, Y  +388.986, Z    +0.000, E1   -15.047, E3 +74694.518}
SPL {X  -162.820, Y  +394.732, Z    +0.000, E1   -28.992, E3 +74694.369}
SPL {X  -162.820, Y  +403.075, Z    +0.000, E1   -46.096, E3 +74694.599}
SPL {X  -162.820, Y  +414.705, Z    +0.000, E1   -61.052, E3 +74694.046}
SPL {X  -162.820, Y  +466.149, Z    +0.000, E1   -74.732, E3 +74704.042}
SPL {X  -160.066, Y  +703.318, Z    +0.000, E1   -76.774, E3 +74788.889}
ENDSPLINE

SPLINE
SPL {X  -161.105, Y  +697.069, Z    +0.000, E1   -74.557, E3 +74810.503}
ENDSPLINE

SPLINE
SPL {X  -159.270, Y  +707.314, Z    +0.000, E1   -74.359, E3 +74818.527}
SPL {X  -156.868, Y  +717.123, Z    +0.000, E1   -74.182, E3 +74826.033}
SPL {X  -153.226, Y  +728.564, Z    +0.000, E1   -73.755, E3 +74837.041}
SPL {X  -149.090, Y  +738.941, Z    +0.000, E1   -73.348, E3 +74846.615}
SPL {X  -145.714, Y  +746.149, Z    +0.000, E1   -72.951, E3 +74854.202}
SPL {X  -140.946, Y  +755.015, Z    +0.000, E1   -72.452, E3 +74863.305}
SPL {X  -136.902, Y  +761.638, Z    +0.000, E1   -71.857, E3 +74871.171}
SPL {X  -133.350, Y  +766.925, Z    +0.000, E1   -71.498, E3 +74876.492}
SPL {X  -129.687, Y  +771.946, Z    +0.000, E1   -71.061, E3 +74881.858}
SPL {X  -126.374, Y  +776.164, Z    +0.000, E1   -70.494, E3 +74887.111}
SPL {X  -123.763, Y  +779.297, Z    +0.000, E1   -70.128, E3 +74890.487}
SPL {X  -119.350, Y  +784.252, Z    +0.000, E1   -71.016, E3 +74889.687}
SPL {X   -61.593, Y  +824.220, Z    +0.000, E1   -55.970, E3 +75056.003}
ENDSPLINE

SPLINE
SPL {X  -131.598, Y  +769.376, Z    +0.000, E1   -56.871, E3 +75222.275}
SPL {X  -152.760, Y  +729.846, Z    +0.000, E1   -44.713, E3 +75229.327}
SPL {X  -158.868, Y  +709.157, Z    +0.000, E1   -33.466, E3 +75230.528}
SPL {X  -161.987, Y  +689.949, Z    +0.000, E1   -18.777, E3 +75231.489}
SPL {X  -162.803, Y  +675.860, Z    +0.000, E1    -4.958, E3 +75231.471}
SPL {X  -162.820, Y  +671.500, Z    +0.000, E1    +0.000, E3 +75231.008}
SPL {X  -162.820, Y  +669.410, Z    +0.000, E1    +4.515, E3 +75230.770}
SPL {X  -162.820, Y  +664.781, Z    +0.000, E1   +16.411, E3 +75230.765}
SPL {X  -162.820, Y  +659.650, Z    +0.000, E1   +29.778, E3 +75230.775}
SPL {X  -162.820, Y  +654.031, Z    +0.000, E1   +42.449, E3 +75230.689}
SPL {X  -162.820, Y  +647.611, Z    +0.000, E1   +52.483, E3 +75231.219}
SPL {X  -162.820, Y  +637.134, Z    +0.000, E1   +65.232, E3 +75229.467}
SPL {X  -162.820, Y  +616.721, Z    +0.000, E1   +72.273, E3 +75233.201}
SPL {X  -162.820, Y  +577.172, Z    +0.000, E1   +75.843, E3 +75243.181}
SPL {X  -159.895, Y  +349.775, Z    +0.000, E1   +76.042, E3 +75334.848}
ENDSPLINE

SPLINE
SPL {X  -160.357, Y  +352.285, Z    +0.000, E1   +74.783, E3 +75347.785}
ENDSPLINE

SPLINE
SPL {X  -145.737, Y  +307.897, Z    +0.000, E1   +77.368, E3 +75340.361}
SPL {X  -145.122, Y  +306.676, Z    +0.000, E1   +76.360, E3 +75351.713}
ENDSPLINE

SPLINE
SPL {X  -145.186, Y  +306.802, Z    +0.000, E1   +74.850, E3 +75366.067}
ENDSPLINE

SPLINE
SPL {X  -143.742, Y  +304.025, Z    +0.000, E1   +73.644, E3 +75378.121}
SPL {X  -141.993, Y  +300.823, Z    +0.000, E1   +72.659, E3 +75387.693}
SPL {X  -138.166, Y  +294.358, Z    +0.000, E1   +72.281, E3 +75394.155}
SPL {X  -134.385, Y  +288.571, Z    +0.000, E1   +71.826, E3 +75400.418}
SPL {X  -129.872, Y  +282.297, Z    +0.000, E1   +71.229, E3 +75407.588}
SPL {X  -124.448, Y  +275.510, Z    +0.000, E1   +70.509, E3 +75414.961}
SPL {X  -117.513, Y  +267.801, Z    +0.000, E1   +72.197, E3 +75412.544}
SPL {X   -63.140, Y  +230.421, Z    +0.000, E1   +55.875, E3 +75581.983}
ENDSPLINE

SPLINE
SPL {X  -130.329, Y  +282.905, Z    +0.000, E1   +55.659, E3 +75740.318}
SPL {X  -154.728, Y  +329.807, Z    +0.000, E1   +40.640, E3 +75749.700}
SPL {X  -160.994, Y  +356.185, Z    +0.000, E1   +24.373, E3 +75752.293}
SPL {X  -162.352, Y  +368.168, Z    +0.000, E1   +14.282, E3 +75752.345}
SPL {X  -162.808, Y  +378.562, Z    +0.000, E1    +4.298, E3 +75752.277}
SPL {X  -162.820, Y  +382.822, Z    +0.000, E1    -0.352, E3 +75751.785}
SPL {X  -162.820, Y  +387.647, Z    +0.000, E1   -11.488, E3 +75751.594}
SPL {X  -162.820, Y  +393.007, Z    +0.000, E1   -25.093, E3 +75751.552}
SPL {X  -162.820, Y  +400.636, Z    +0.000, E1   -41.711, E3 +75751.602}
SPL {X  -162.820, Y  +414.705, Z    +0.000, E1   -61.052, E3 +75751.188}
SPL {X  -162.820, Y  +466.149, Z    +0.000, E1   -74.732, E3 +75761.185}
SPL {X  -160.066, Y  +703.318, Z    +0.000, E1   -76.774, E3 +75846.032}
ENDSPLINE

SPLINE
SPL {X  -161.105, Y  +697.069, Z    +0.000, E1   -74.557, E3 +75867.646}
ENDSPLINE

SPLINE
SPL {X  -159.270, Y  +707.314, Z    +0.000, E1   -74.359, E3 +75875.670}
SPL {X  -156.868, Y  +717.123, Z    +0.000, E1   -74.182, E3 +75883.176}
SPL {X  -153.226, Y  +728.564, Z    +0.000, E1   -73.755, E3 +75894.184}
SPL {X  -149.090, Y  +738.941, Z    +0.000, E1   -73.348, E3 +75903.758}
SPL {X  -145.714, Y  +746.149, Z    +0.000, E1   -72.951, E3 +75911.345}
SPL {X  -142.592, Y  +752.100, Z    +0.000, E1   -72.554, E3 +75917.877}
SPL {X  -139.608, Y  +757.285, Z    +0.000, E1   -72.326, E3 +75922.547}
SPL {X  -136.902, Y  +761.638, Z    +0.000, E1   -71.857, E3 +75928.314}
SPL {X  -133.350, Y  +766.925, Z    +0.000, E1   -71.498, E3 +75933.635}
SPL {X  -129.687, Y  +771.946, Z    +0.000, E1   -71.061, E3 +75939.001}
SPL {X  -126.374, Y  +776.164, Z    +0.000, E1   -70.494, E3 +75944.254}
SPL {X  -123.763, Y  +779.297, Z    +0.000, E1   -70.128, E3 +75947.630}
SPL {X  -119.350, Y  +784.252, Z    +0.000, E1   -71.016, E3 +75946.830}
SPL {X   -61.593, Y  +824.220, Z    +0.000, E1   -55.970, E3 +76113.146}
ENDSPLINE

SPLINE
SPL {X  -131.598, Y  +769.376, Z    +0.000, E1   -56.871, E3 +76279.418}
SPL {X  -152.760, Y  +729.846, Z    +0.000, E1   -44.713, E3 +76286.470}
SPL {X  -158.868, Y  +709.157, Z    +0.000, E1   -33.466, E3 +76287.671}
SPL {X  -161.987, Y  +689.949, Z    +0.000, E1   -18.777, E3 +76288.632}
SPL {X  -162.803, Y  +675.860, Z    +0.000, E1    -4.958, E3 +76288.614}
SPL {X  -162.820, Y  +671.500, Z    +0.000, E1    +0.000, E3 +76288.151}
SPL {X  -162.820, Y  +669.410, Z    +0.000, E1    +4.515, E3 +76287.913}
SPL {X  -162.820, Y  +664.781, Z    +0.000, E1   +16.411, E3 +76287.908}
SPL {X  -162.820, Y  +659.650, Z    +0.000, E1   +29.778, E3 +76287.918}
SPL {X  -162.820, Y  +654.031, Z    +0.000, E1   +42.449, E3 +76287.832}
SPL {X  -162.820, Y  +647.611, Z    +0.000, E1   +52.483, E3 +76288.362}
SPL {X  -162.820, Y  +633.243, Z    +0.000, E1   +67.111, E3 +76287.323}
SPL {X  -162.820, Y  +577.172, Z    +0.000, E1   +75.843, E3 +76300.324}
SPL {X  -159.895, Y  +349.775, Z    +0.000, E1   +76.042, E3 +76391.990}
ENDSPLINE

SPLINE
SPL {X  -160.357, Y  +352.285, Z    +0.000, E1   +74.783, E3 +76404.928}
ENDSPLINE

SPLINE
SPL {X  -145.737, Y  +307.897, Z    +0.000, E1   +77.368, E3 +76397.503}
SPL {X  -145.329, Y  +307.084, Z    +0.000, E1   +76.571, E3 +76406.340}
ENDSPLINE

SPLINE
SPL {X  -145.355, Y  +307.136, Z    +0.000, E1   +75.607, E3 +76415.864}
ENDSPLINE

SPLINE
SPL {X  -144.515, Y  +305.495, Z    +0.000, E1   +74.543, E3 +76426.673}
SPL {X  -143.690, Y  +303.925, Z    +0.000, E1   +73.372, E3 +76437.412}
SPL {X  -141.993, Y  +300.823, Z    +0.000, E1   +72.659, E3 +76444.836}
SPL {X  -138.166, Y  +294.358, Z    +0.000, E1   +72.281, E3 +76451.297}
SPL {X  -134.385, Y  +288.571, Z    +0.000, E1   +71.826, E3 +76457.561}
SPL {X  -130.773, Y  +283.501, Z    +0.000, E1   +71.398, E3 +76462.985}
SPL {X  -126.922, Y  +278.513, Z    +0.000, E1   +70.767, E3 +76469.139}
SPL {X  -123.520, Y  +274.419, Z    +0.000, E1   +70.342, E3 +76473.338}
SPL {X  -117.513, Y  +267.801, Z    +0.000, E1   +72.197, E3 +76469.687}
SPL {X   -63.140, Y  +230.421, Z    +0.000, E1   +55.875, E3 +76639.125}
ENDSPLINE

SPLINE
SPL {X  -130.329, Y  +282.905, Z    +0.000, E1   +55.659, E3 +76797.461}
SPL {X  -154.728, Y  +329.807, Z    +0.000, E1   +40.640, E3 +76806.843}
SPL {X  -160.994, Y  +356.185, Z    +0.000, E1   +24.373, E3 +76809.435}
SPL {X  -162.352, Y  +368.168, Z    +0.000, E1   +14.282, E3 +76809.488}
SPL {X  -162.808, Y  +378.562, Z    +0.000, E1    +4.298, E3 +76809.420}
SPL {X  -162.820, Y  +382.500, Z    +0.000, E1    +0.000, E3 +76808.993}
SPL {X  -162.820, Y  +384.915, Z    +0.000, E1    -4.894, E3 +76808.706}
SPL {X  -162.820, Y  +388.986, Z    +0.000, E1   -15.047, E3 +76808.804}
SPL {X  -162.820, Y  +393.007, Z    +0.000, E1   -25.093, E3 +76808.695}
SPL {X  -162.820, Y  +400.636, Z    +0.000, E1   -41.711, E3 +76808.745}
SPL {X  -162.820, Y  +414.705, Z    +0.000, E1   -61.052, E3 +76808.331}
SPL {X  -162.820, Y  +466.149, Z    +0.000, E1   -74.732, E3 +76818.327}
SPL {X  -160.066, Y  +703.318, Z    +0.000, E1   -76.774, E3 +76903.175}
ENDSPLINE

SPLINE
SPL {X  -161.105, Y  +697.069, Z    +0.000, E1   -74.557, E3 +76924.789}
ENDSPLINE

SPLINE
SPL {X  -159.270, Y  +707.314, Z    +0.000, E1   -74.359, E3 +76932.813}
SPL {X  -156.868, Y  +717.123, Z    +0.000, E1   -74.182, E3 +76940.319}
SPL {X  -153.226, Y  +728.564, Z    +0.000, E1   -73.755, E3 +76951.327}
SPL {X  -149.090, Y  +738.941, Z    +0.000, E1   -73.348, E3 +76960.901}
SPL {X  -145.714, Y  +746.149, Z    +0.000, E1   -72.951, E3 +76968.487}
SPL {X  -140.946, Y  +755.015, Z    +0.000, E1   -72.452, E3 +76977.590}
SPL {X  -136.902, Y  +761.638, Z    +0.000, E1   -71.857, E3 +76985.457}
SPL {X  -133.350, Y  +766.925, Z    +0.000, E1   -71.498, E3 +76990.778}
SPL {X  -129.687, Y  +771.946, Z    +0.000, E1   -71.061, E3 +76996.144}
SPL {X  -126.374, Y  +776.164, Z    +0.000, E1   -70.494, E3 +77001.397}
SPL {X  -123.763, Y  +779.297, Z    +0.000, E1   -70.128, E3 +77004.773}
SPL {X  -119.350, Y  +784.252, Z    +0.000, E1   -71.016, E3 +77003.973}
SPL {X   -61.593, Y  +824.220, Z    +0.000, E1   -55.970, E3 +77170.289}
ENDSPLINE

SPLINE
SPL {X  -131.598, Y  +769.376, Z    +0.000, E1   -56.871, E3 +77336.560}
SPL {X  -152.760, Y  +729.846, Z    +0.000, E1   -44.713, E3 +77343.613}
SPL {X  -158.868, Y  +709.157, Z    +0.000, E1   -33.466, E3 +77344.814}
SPL {X  -161.987, Y  +689.949, Z    +0.000, E1   -18.777, E3 +77345.775}
SPL {X  -162.803, Y  +675.860, Z    +0.000, E1    -4.958, E3 +77345.757}
SPL {X  -162.820, Y  +671.500, Z    +0.000, E1    +0.000, E3 +77345.293}
SPL {X  -162.820, Y  +669.410, Z    +0.000, E1    +4.515, E3 +77345.056}
SPL {X  -162.820, Y  +664.781, Z    +0.000, E1   +16.411, E3 +77345.051}
SPL {X  -162.820, Y  +659.650, Z    +0.000, E1   +29.778, E3 +77345.061}
SPL {X  -162.820, Y  +654.031, Z    +0.000, E1   +42.449, E3 +77344.975}
SPL {X  -162.820, Y  +647.611, Z    +0.000, E1   +52.483, E3 +77345.505}
SPL {X  -162.820, Y  +633.243, Z    +0.000, E1   +67.111, E3 +77344.465}
SPL {X  -162.820, Y  +577.172, Z    +0.000, E1   +75.843, E3 +77357.467}
SPL {X  -159.895, Y  +349.775, Z    +0.000, E1   +76.042, E3 +77449.133}
ENDSPLINE

SPLINE
SPL {X  -160.357, Y  +352.285, Z    +0.000, E1   +74.783, E3 +77462.071}
ENDSPLINE

SPLINE
SPL {X  -145.737, Y  +307.897, Z    +0.000, E1   +77.368, E3 +77454.646}
SPL {X  -145.329, Y  +307.084, Z    +0.000, E1   +76.571, E3 +77463.482}
ENDSPLINE

SPLINE
SPL {X  -145.355, Y  +307.136, Z    +0.000, E1   +75.607, E3 +77473.007}
ENDSPLINE

SPLINE
SPL {X  -144.515, Y  +305.495, Z    +0.000, E1   +74.543, E3 +77483.816}
SPL {X  -143.690, Y  +303.925, Z    +0.000, E1   +73.372, E3 +77494.554}
SPL {X  -141.993, Y  +300.823, Z    +0.000, E1   +72.659, E3 +77501.979}
SPL {X  -138.166, Y  +294.358, Z    +0.000, E1   +72.281, E3 +77508.440}
SPL {X  -134.385, Y  +288.571, Z    +0.000, E1   +71.826, E3 +77514.704}
SPL {X  -130.773, Y  +283.501, Z    +0.000, E1   +71.398, E3 +77520.128}
SPL {X  -126.922, Y  +278.513, Z    +0.000, E1   +70.767, E3 +77526.282}
SPL {X  -123.520, Y  +274.419, Z    +0.000, E1   +70.342, E3 +77530.481}
SPL {X  -117.513, Y  +267.801, Z    +0.000, E1   +72.197, E3 +77526.830}
SPL {X   -63.140, Y  +230.421, Z    +0.000, E1   +55.875, E3 +77696.268}
ENDSPLINE

SPLINE
SPL {X  -130.329, Y  +282.905, Z    +0.000, E1   +55.659, E3 +77854.604}
SPL {X  -154.728, Y  +329.807, Z    +0.000, E1   +40.640, E3 +77863.985}
SPL {X  -160.994, Y  +356.185, Z    +0.000, E1   +24.373, E3 +77866.578}
SPL {X  -162.352, Y  +368.168, Z    +0.000, E1   +14.282, E3 +77866.631}
SPL {X  -162.808, Y  +378.562, Z    +0.000, E1    +4.298, E3 +77866.563}
SPL {X  -162.820, Y  +382.500, Z    +0.000, E1    +0.000, E3 +77866.136}
SPL {X  -162.820, Y  +384.915, Z    +0.000, E1    -4.894, E3 +77865.849}
SPL {X  -162.820, Y  +388.986, Z    +0.000, E1   -15.047, E3 +77865.947}
SPL {X  -162.820, Y  +393.007, Z    +0.000, E1   -25.093, E3 +77865.838}
SPL {X  -162.820, Y  +400.636, Z    +0.000, E1   -41.711, E3 +77865.888}
SPL {X  -162.820, Y  +414.705, Z    +0.000, E1   -61.052, E3 +77865.474}
SPL {X  -162.820, Y  +466.149, Z    +0.000, E1   -74.732, E3 +77875.470}
SPL {X  -160.722, Y  +699.554, Z    +0.000, E1   -75.485, E3 +77972.880}
SPL {X  -159.966, Y  +703.854, Z    +0.000, E1   -74.386, E3 +77987.784}
SPL {X  -156.868, Y  +717.123, Z    +0.000, E1   -74.182, E3 +77997.462}
SPL {X  -153.226, Y  +728.564, Z    +0.000, E1   -73.755, E3 +78008.470}
SPL {X  -149.090, Y  +738.941, Z    +0.000, E1   -73.348, E3 +78018.043}
SPL {X  -145.714, Y  +746.149, Z    +0.000, E1   -72.951, E3 +78025.630}
SPL {X  -140.946, Y  +755.015, Z    +0.000, E1   -72.452, E3 +78034.733}
SPL {X  -136.902, Y  +761.638, Z    +0.000, E1   -71.857, E3 +78042.600}
SPL {X  -133.350, Y  +766.925, Z    +0.000, E1   -71.498, E3 +78047.920}
SPL {X  -129.687, Y  +771.946, Z    +0.000, E1   -71.061, E3 +78053.286}
SPL {X  -126.374, Y  +776.164, Z    +0.000, E1   -70.494, E3 +78058.540}
SPL {X  -123.763, Y  +779.297, Z    +0.000, E1   -70.128, E3 +78061.916}
SPL {X  -119.350, Y  +784.252, Z    +0.000, E1   -71.016, E3 +78061.116}
SPL {X   -61.593, Y  +824.220, Z    +0.000, E1   -55.970, E3 +78227.431}
ENDSPLINE

SPLINE
SPL {X  -131.598, Y  +769.376, Z    +0.000, E1   -56.871, E3 +78393.703}
SPL {X  -152.760, Y  +729.846, Z    +0.000, E1   -44.713, E3 +78400.756}
SPL {X  -158.868, Y  +709.157, Z    +0.000, E1   -33.466, E3 +78401.957}
SPL {X  -161.987, Y  +689.949, Z    +0.000, E1   -18.777, E3 +78402.918}
SPL {X  -162.803, Y  +675.860, Z    +0.000, E1    -4.958, E3 +78402.900}
SPL {X  -162.820, Y  +671.500, Z    +0.000, E1    +0.000, E3 +78402.436}
SPL {X  -162.820, Y  +669.410, Z    +0.000, E1    +4.515, E3 +78402.198}
SPL {X  -162.820, Y  +664.781, Z    +0.000, E1   +16.411, E3 +78402.194}
SPL {X  -162.820, Y  +659.650, Z    +0.000, E1   +29.778, E3 +78402.204}
SPL {X  -162.820, Y  +654.031, Z    +0.000, E1   +42.449, E3 +78402.117}
SPL {X  -162.820, Y  +647.611, Z    +0.000, E1   +52.483, E3 +78402.648}
SPL {X  -162.820, Y  +637.134, Z    +0.000, E1   +65.232, E3 +78400.896}
SPL {X  -162.820, Y  +616.721, Z    +0.000, E1   +72.273, E3 +78404.630}
SPL {X  -162.820, Y  +577.172, Z    +0.000, E1   +75.843, E3 +78414.610}
SPL {X  -159.895, Y  +349.775, Z    +0.000, E1   +76.042, E3 +78506.276}
ENDSPLINE

SPLINE
SPL {X  -160.357, Y  +352.285, Z    +0.000, E1   +74.783, E3 +78519.214}
ENDSPLINE

SPLINE
SPL {X  -145.737, Y  +307.897, Z    +0.000, E1   +77.368, E3 +78511.789}
SPL {X  -145.122, Y  +306.676, Z    +0.000, E1   +76.360, E3 +78523.142}
ENDSPLINE

SPLINE
SPL {X  -145.186, Y  +306.802, Z    +0.000, E1   +74.850, E3 +78537.495}
ENDSPLINE

SPLINE
SPL {X  -143.742, Y  +304.025, Z    +0.000, E1   +73.644, E3 +78549.550}
SPL {X  -141.993, Y  +300.823, Z    +0.000, E1   +72.659, E3 +78559.122}
SPL {X  -138.166, Y  +294.358, Z    +0.000, E1   +72.281, E3 +78565.583}
SPL {X  -134.385, Y  +288.571, Z    +0.000, E1   +71.826, E3 +78571.847}
SPL {X  -129.872, Y  +282.297, Z    +0.000, E1   +71.229, E3 +78579.017}
SPL {X  -124.448, Y  +275.510, Z    +0.000, E1   +70.509, E3 +78586.390}
SPL {X  -117.513, Y  +267.801, Z    +0.000, E1   +72.197, E3 +78583.972}
SPL {X   -63.140, Y  +230.421, Z    +0.000, E1   +55.875, E3 +78753.411}
ENDSPLINE

SPLINE
SPL {X  -130.329, Y  +282.905, Z    +0.000, E1   +55.659, E3 +78911.747}
SPL {X  -154.728, Y  +329.807, Z    +0.000, E1   +40.640, E3 +78921.128}
SPL {X  -160.994, Y  +356.185, Z    +0.000, E1   +24.373, E3 +78923.721}
SPL {X  -162.637, Y  +372.778, Z    +0.000, E1   +10.098, E3 +78923.741}
SPL {X  -162.820, Y  +382.419, Z    +0.000, E1    +0.163, E3 +78923.301}
SPL {X  -162.820, Y  +384.915, Z    +0.000, E1    -4.894, E3 +78922.992}
SPL {X  -162.820, Y  +388.986, Z    +0.000, E1   -15.047, E3 +78923.090}
SPL {X  -162.820, Y  +394.732, Z    +0.000, E1   -28.992, E3 +78922.941}
SPL {X  -162.820, Y  +403.075, Z    +0.000, E1   -46.096, E3 +78923.171}
SPL {X  -162.820, Y  +414.705, Z    +0.000, E1   -61.052, E3 +78922.617}
SPL {X  -162.820, Y  +466.149, Z    +0.000, E1   -74.732, E3 +78932.613}
SPL {X  -160.066, Y  +703.318, Z    +0.000, E1   -76.774, E3 +79017.461}
ENDSPLINE

SPLINE
SPL {X  -161.105, Y  +697.069, Z    +0.000, E1   -74.557, E3 +79039.075}
ENDSPLINE

SPLINE
SPL {X  -159.270, Y  +707.314, Z    +0.000, E1   -74.359, E3 +79047.099}
SPL {X  -156.868, Y  +717.123, Z    +0.000, E1   -74.182, E3 +79054.605}
SPL {X  -153.226, Y  +728.564, Z    +0.000, E1   -73.755, E3 +79065.613}
SPL {X  -149.090, Y  +738.941, Z    +0.000, E1   -73.348, E3 +79075.186}
SPL {X  -145.714, Y  +746.149, Z    +0.000, E1   -72.951, E3 +79082.773}
SPL {X  -140.946, Y  +755.015, Z    +0.000, E1   -72.452, E3 +79091.876}
SPL {X  -136.902, Y  +761.638, Z    +0.000, E1   -71.857, E3 +79099.743}
SPL {X  -133.350, Y  +766.925, Z    +0.000, E1   -71.498, E3 +79105.063}
SPL {X  -129.687, Y  +771.946, Z    +0.000, E1   -71.061, E3 +79110.429}
SPL {X  -126.374, Y  +776.164, Z    +0.000, E1   -70.494, E3 +79115.683}
SPL {X  -123.763, Y  +779.297, Z    +0.000, E1   -70.128, E3 +79119.059}
SPL {X  -119.350, Y  +784.252, Z    +0.000, E1   -71.016, E3 +79118.259}
SPL {X   -61.593, Y  +824.220, Z    +0.000, E1   -55.970, E3 +79284.574}
ENDSPLINE

